HMI tags "ProLav1"
   "Lav1_Prog1_EnjIni_Cant" : Int AT 4x402562, 10 min
   "Lav1_Prog1_EnjIni_NivAg" : Int AT 4x402563, 10 min
   "Lav1_Prog1_EnjIni_Tiempo" : Int AT 4x402564, 10 min
   "Lav1_Prog1_PreLav_NivAg" : Int AT 4x402566, 10 min
   "Lav1_Prog1_PreLav_AgCaliente" : Int AT 4x402567, 10 min
   "Lav1_Prog1_Lav1_NivAg" : Int AT 4x402569, 10 min
   "Lav1_Prog1_Lav1_AgCaliente" : Int AT 4x402570, 10 min
   "Lav1_Prog1_EnjFin_Cant" : Int AT 4x402571, 10 s
   "Lav1_Prog1_Lav2_Tiempo" : Int AT 4x402617, 10 min
   "Lav1_Prog1_Lav2_NivAg" : Int AT 4x402572, 10 min
   "Lav1_Prog1_EnjFin_Tiempo" : Int AT 4x402573, 10 min
   "Lav1_Prog1_Lav2_AgCaliente" : Int AT 4x402574, 10 min
   "Lav1_Prog1_Centr_Tiempo" : Int AT 4x402575, 10 min
   "Lav1_Prog1_PreLav_Vapor" : Int AT 4x402576, 10 min
   "Lav1_Prog1_PreLav_Temperatura" : Int AT 4x402589, 10 min
   "Lav1_Prog1_Lav1_Temperatura" : Int AT 4x402591, 10 min
   "Lav1_Prog1_Lav2_Temperatura" : Int AT 4x401057, 10 min
   "Lav1_Prog1_PreLav_Tiempo" : Int AT 4x402565, 10 min
   "Lav1_Prog1_Lav1_Tiempo" : Int AT 4x402568, 10 min
   "Lav1_Prog2_EnjIni_Cant" : Int AT 4x402626, 10 min
   "Lav1_Prog2_EnjIni_NivAg" : Int AT 4x402627, 10 min
   "Lav1_Prog2_EnjIni_Tiempo" : Int AT 4x402628, 10 min
   "Lav1_Prog2_PreLav_NivAg" : Int AT 4x402630, 10 min
   "Lav1_Prog2_PreLav_AgCaliente" : Int AT 4x402631, 10 min
   "Lav1_Prog2_Lav1_NivAg" : Int AT 4x402633, 10 min
   "Lav1_Prog2_Lav1_AgCaliente" : Int AT 4x402634, 10 min
   "Lav1_Prog2_EnjFin_Cant" : Int AT 4x402635, 10 s
   "Lav1_Prog2_Lav2_Tiempo" : Int AT 4x402618, 10 min
   "Lav1_Prog2_Lav2_NivAg" : Int AT 4x402636, 10 min
   "Lav1_Prog2_EnjFin_Tiempo" : Int AT 4x402637, 10 min
   "Lav1_Prog2_Lav2_AgCaliente" : Int AT 4x402638, 10 min
   "Lav1_Prog2_Centr_Tiempo" : Int AT 4x402639, 10 min
   "Lav1_Prog2_PreLav_Vapor" : Int AT 4x402577, 10 min
   "Lav1_Prog2_PreLav_Temperatura" : Int AT 4x402592, 10 min
   "Lav1_Prog2_Lav1_Temperatura" : Int AT 4x402593, 10 min
   "Lav1_Prog2_Lav2_Temperatura" : Int AT 4x401058, 10 min
   "Lav1_Prog2_PreLav_Tiempo" : Int AT 4x402629, 10 min
   "Lav1_Prog2_Lav1_Tiempo" : Int AT 4x402632, 10 min
   "Lav1_Prog3_EnjIni_Cant" : Int AT 4x402690, 10 s
   "Lav1_Prog3_EnjIni_NivAg" : Int AT 4x402691, 10 min
   "Lav1_Prog3_EnjIni_Tiempo" : Int AT 4x402692, 10 min
   "Lav1_Prog3_PreLav_NivAg" : Int AT 4x402694, 10 min
   "Lav1_Prog3_PreLav_AgCaliente" : Int AT 4x402695, 10 min
   "Lav1_Prog3_Lav1_NivAg" : Int AT 4x402697, 10 min
   "Lav1_Prog3_Lav1_AgCaliente" : Int AT 4x402698, 10 min
   "Lav1_Prog3_EnjFin_Cant" : Int AT 4x402699, 10 min
   "Lav1_Prog3_Lav2_Tiempo" : Int AT 4x402619, 10 min
   "Lav1_Prog3_Lav2_NivAg" : Int AT 4x402700, 10 min
   "Lav1_Prog3_EnjFin_Tiempo" : Int AT 4x402701, 10 min
   "Lav1_Prog3_Lav2_AgCaliente" : Int AT 4x402702, 10 min
   "Lav1_Prog3_Centr_Tiempo" : Int AT 4x402703, 10 min
   "Lav1_Prog3_PreLav_Vapor" : Int AT 4x402579, 10 min
   "Lav1_Prog3_PreLav_Temperatura" : Int AT 4x402595, 10 min
   "Lav1_Prog3_Lav1_Temperatura" : Int AT 4x402597, 10 min
   "Lav1_Prog3_Lav2_Temperatura" : Int AT 4x401059, 10 min
   "Lav1_Prog3_PreLav_Tiempo" : Int AT 4x402693, 10 min
   "Lav1_Prog3_Lav1_Tiempo" : Int AT 4x402696, 10 min
   "Lav1_Prog4_EnjIni_Cant" : Int AT 4x402754, 10 s
   "Lav1_Prog4_EnjIni_NivAg" : Int AT 4x402755, 10 min
   "Lav1_Prog4_EnjIni_Tiempo" : Int AT 4x402756, 10 min
   "Lav1_Prog4_PreLav_NivAg" : Int AT 4x402758, 10 min
   "Lav1_Prog4_PreLav_AgCaliente" : Int AT 4x402759, 10 min
   "Lav1_Prog4_Lav1_NivAg" : Int AT 4x402761, 10 min
   "Lav1_Prog4_Lav1_AgCaliente" : Int AT 4x402762, 10 min
   "Lav1_Prog4_EnjFin_Cant" : Int AT 4x402763, 10 min
   "Lav1_Prog4_Lav2_Tiempo" : Int AT 4x402620, 10 min
   "Lav1_Prog4_Lav2_NivAg" : Int AT 4x402764, 10 min
   "Lav1_Prog4_EnjFin_Tiempo" : Int AT 4x402765, 10 min
   "Lav1_Prog4_Lav2_AgCaliente" : Int AT 4x402766, 10 min
   "Lav1_Prog4_Centr_Tiempo" : Int AT 4x402767, 10 min
   "Lav1_Prog4_PreLav_Vapor" : Int AT 4x402581, 10 min
   "Lav1_Prog4_PreLav_Temperatura" : Int AT 4x402599, 10 min
   "Lav1_Prog4_Lav1_Temperatura" : Int AT 4x402600, 10 min
   "Lav1_Prog4_Lav2_Temperatura" : Int AT 4x401060, 10 min
   "Lav1_Prog4_PreLav_Tiempo" : Int AT 4x402757, 10 min
   "Lav1_Prog4_Lav1_Tiempo" : Int AT 4x402760, 10 min
   "Lav1_Prog5_EnjIni_Cant" : Int AT 4x402818, 10 min
   "Lav1_Prog5_EnjIni_NivAg" : Int AT 4x402819, 10 min
   "Lav1_Prog5_EnjIni_Tiempo" : Int AT 4x402820, 10 min
   "Lav1_Prog5_PreLav_NivAg" : Int AT 4x402822, 10 min
   "Lav1_Prog5_PreLav_AgCaliente" : Int AT 4x402823, 10 min
   "Lav1_Prog5_Lav1_NivAg" : Int AT 4x402825, 10 min
   "Lav1_Prog5_Lav1_AgCaliente" : Int AT 4x402826, 10 min
   "Lav1_Prog5_EnjFin_Cant" : Int AT 4x402827, 10 s
   "Lav1_Prog5_Lav2_Tiempo" : Int AT 4x402621, 10 min
   "Lav1_Prog5_Lav2_NivAg" : Int AT 4x402828, 10 min
   "Lav1_Prog5_EnjFin_Tiempo" : Int AT 4x402829, 10 min
   "Lav1_Prog5_Lav2_AgCaliente" : Int AT 4x402830, 10 min
   "Lav1_Prog5_Centr_Tiempo" : Int AT 4x402831, 10 min
   "Lav1_Prog5_PreLav_Vapor" : Int AT 4x402583, 10 min
   "Lav1_Prog5_PreLav_Temperatura" : Int AT 4x402601, 10 min
   "Lav1_Prog5_Lav1_Temperatura" : Int AT 4x402603, 10 min
   "Lav1_Prog5_Lav2_Temperatura" : Int AT 4x401061, 10 min
   "Lav1_Prog5_PreLav_Tiempo" : Int AT 4x402821, 10 min
   "Lav1_Prog5_Lav1_Tiempo" : Int AT 4x402824, 10 min
   "Lav1_Prog6_EnjIni_Cant" : Int AT 4x402882, 10 min
   "Lav1_Prog6_EnjIni_NivAg" : Int AT 4x402883, 10 min
   "Lav1_Prog6_EnjIni_Tiempo" : Int AT 4x402884, 10 min
   "Lav1_Prog6_PreLav_NivAg" : Int AT 4x402886, 10 min
   "Lav1_Prog6_PreLav_AgCaliente" : Int AT 4x402887, 10 min
   "Lav1_Prog6_Lav1_NivAg" : Int AT 4x402889, 10 min
   "Lav1_Prog6_Lav1_AgCaliente" : Int AT 4x402890, 10 min
   "Lav1_Prog6_EnjFin_Cant" : Int AT 4x402891, 10 s
   "Lav1_Prog6_Lav2_Tiempo" : Int AT 4x402622, 10 min
   "Lav1_Prog6_Lav2_NivAg" : Int AT 4x402892, 10 min
   "Lav1_Prog6_EnjFin_Tiempo" : Int AT 4x402893, 10 min
   "Lav1_Prog6_Lav2_AgCaliente" : Int AT 4x402894, 10 min
   "Lav1_Prog6_Centr_Tiempo" : Int AT 4x402895, 10 min
   "Lav1_Prog6_PreLav_Vapor" : Int AT 4x402585, 10 min
   "Lav1_Prog6_PreLav_Temperatura" : Int AT 4x402605, 10 min
   "Lav1_Prog6_Lav1_Temperatura" : Int AT 4x402607, 10 min
   "Lav1_Prog6_Lav2_Temperatura" : Int AT 4x401062, 10 min
   "Lav1_Prog6_PreLav_Tiempo" : Int AT 4x402885, 10 min
   "Lav1_Prog6_Lav1_Tiempo" : Int AT 4x402888, 10 min
   "Lav1_Prog7_EnjIni_Cant" : Int AT 4x402953, 10 s
   "Lav1_Prog7_EnjIni_NivAg" : Int AT 4x402955, 10 min
   "Lav1_Prog7_EnjIni_Tiempo" : Int AT 4x402956, 10 min
   "Lav1_Prog7_PreLav_NivAg" : Int AT 4x402958, 10 min
   "Lav1_Prog7_PreLav_AgCaliente" : Int AT 4x402959, 10 min
   "Lav1_Prog7_Lav1_NivAg" : Int AT 4x402961, 10 min
   "Lav1_Prog7_Lav1_AgCaliente" : Int AT 4x402962, 10 min
   "Lav1_Prog7_EnjFin_Cant" : Int AT 4x402964, 10 min
   "Lav1_Prog7_Lav2_Tiempo" : Int AT 4x402963, 10 min
   "Lav1_Prog7_Lav2_NivAg" : Int AT 4x402965, 10 min
   "Lav1_Prog7_EnjFin_Tiempo" : Int AT 4x402966, 10 min
   "Lav1_Prog7_Lav2_AgCaliente" : Int AT 4x402967, 10 min
   "Lav1_Prog7_Centr_Tiempo" : Int AT 4x402968, 10 min
   "Lav1_Prog7_PreLav_Vapor" : Int AT 4x402969, 10 min
   "Lav1_Prog7_PreLav_Temperatura" : Int AT 4x402970, 10 min
   "Lav1_Prog7_Lav1_Temperatura" : Int AT 4x402971, 10 min
   "Lav1_Prog7_Lav2_Temperatura" : Int AT 4x401121, 10 min
   "Lav1_Prog7_PreLav_Tiempo" : Int AT 4x402957, 10 min
   "Lav1_Prog7_Lav1_Tiempo" : Int AT 4x402960, 10 min
   "Lav1_Prog8_EnjIni_Cant" : Int AT 4x402978, 10 min
   "Lav1_Prog8_EnjIni_NivAg" : Int AT 4x402979, 10 min
   "Lav1_Prog8_EnjIni_Tiempo" : Int AT 4x402980, 10 min
   "Lav1_Prog8_PreLav_NivAg" : Int AT 4x402982, 10 min
   "Lav1_Prog8_PreLav_AgCaliente" : Int AT 4x402983, 10 min
   "Lav1_Prog8_Lav1_NivAg" : Int AT 4x402985, 10 min
   "Lav1_Prog8_Lav1_AgCaliente" : Int AT 4x402986, 10 min
   "Lav1_Prog8_EnjFin_Cant" : Int AT 4x402988, 10 s
   "Lav1_Prog8_Lav2_Tiempo" : Int AT 4x402987, 10 min
   "Lav1_Prog8_Lav2_NivAg" : Int AT 4x402989, 10 min
   "Lav1_Prog8_EnjFin_Tiempo" : Int AT 4x402990, 10 min
   "Lav1_Prog8_Lav2_AgCaliente" : Int AT 4x402991, 10 min
   "Lav1_Prog8_Centr_Tiempo" : Int AT 4x402992, 10 min
   "Lav1_Prog8_PreLav_Vapor" : Int AT 4x402993, 10 min
   "Lav1_Prog8_PreLav_Temperatura" : Int AT 4x402994, 10 min
   "Lav1_Prog8_Lav1_Temperatura" : Int AT 4x402995, 10 min
   "Lav1_Prog8_Lav2_Temperatura" : Int AT 4x401186, 10 min
   "Lav1_Prog8_PreLav_Tiempo" : Int AT 4x402981, 10 min
   "Lav1_Prog8_Lav1_Tiempo" : Int AT 4x402984, 10 min
   "Lav1_Prog9_EnjIni_Cant" : Int AT 4x402996, 10 min
   "Lav1_Prog9_EnjIni_NivAg" : Int AT 4x402997, 10 min
   "Lav1_Prog9_EnjIni_Tiempo" : Int AT 4x402998, 10 min
   "Lav1_Prog9_PreLav_NivAg" : Int AT 4x403000, 10 min
   "Lav1_Prog9_PreLav_AgCaliente" : Int AT 4x403001, 10 min
   "Lav1_Prog9_Lav1_NivAg" : Int AT 4x403003, 10 min
   "Lav1_Prog9_Lav1_AgCaliente" : Int AT 4x403004, 10 min
   "Lav1_Prog9_EnjFin_Cant" : Int AT 4x403006, 10 s
   "Lav1_Prog9_Lav2_Tiempo" : Int AT 4x403005, 10 min
   "Lav1_Prog9_Lav2_NivAg" : Int AT 4x403007, 10 min
   "Lav1_Prog9_EnjFin_Tiempo" : Int AT 4x403008, 10 min
   "Lav1_Prog9_Lav2_AgCaliente" : Int AT 4x403009, 10 min
   "Lav1_Prog9_Centr_Tiempo" : Int AT 4x403010, 10 min
   "Lav1_Prog9_PreLav_Vapor" : Int AT 4x403011, 10 min
   "Lav1_Prog9_PreLav_Temperatura" : Int AT 4x403012, 10 min
   "Lav1_Prog9_Lav1_Temperatura" : Int AT 4x403013, 10 min
   "Lav1_Prog9_Lav2_Temperatura" : Int AT 4x401251, 10 min
   "Lav1_Prog9_PreLav_Tiempo" : Int AT 4x402999, 10 min
   "Lav1_Prog9_Lav1_Tiempo" : Int AT 4x403002, 10 min
   "Lav1_Prog10_EnjIni_Cant" : Int AT 4x403014, 10 min
   "Lav1_Prog10_EnjIni_NivAg" : Int AT 4x403015, 10 min
   "Lav1_Prog10_EnjIni_Tiempo" : Int AT 4x403016, 10 min
   "Lav1_Prog10_PreLav_NivAg" : Int AT 4x403018, 10 min
   "Lav1_Prog10_PreLav_AgCaliente" : Int AT 4x403019, 10 min
   "Lav1_Prog10_Lav1_NivAg" : Int AT 4x403021, 10 min
   "Lav1_Prog10_Lav1_AgCaliente" : Int AT 4x403022, 10 min
   "Lav1_Prog10_EnjFin_Cant" : Int AT 4x403024, 10 s
   "Lav1_Prog10_Lav2_Tiempo" : Int AT 4x403023, 10 min
   "Lav1_Prog10_Lav2_NivAg" : Int AT 4x403025, 10 min
   "Lav1_Prog10_EnjFin_Tiempo" : Int AT 4x403026, 10 min
   "Lav1_Prog10_Lav2_AgCaliente" : Int AT 4x403027, 10 min
   "Lav1_Prog10_Centr_Tiempo" : Int AT 4x403028, 10 min
   "Lav1_Prog10_PreLav_Vapor" : Int AT 4x403029, 10 min
   "Lav1_Prog10_PreLav_Temperatura" : Int AT 4x403030, 10 min
   "Lav1_Prog10_Lav1_Temperatura" : Int AT 4x403031, 10 min
   "Lav1_Prog10_Lav2_Temperatura" : Int AT 4x401316, 10 min
   "Lav1_Prog10_PreLav_Tiempo" : Int AT 4x403017, 10 min
   "Lav1_Prog10_Lav1_Tiempo" : Int AT 4x403020, 10 min
   "Lav1_Prog11_EnjIni_Cant" : Int AT 4x403033, 10 min
   "Lav1_Prog11_EnjIni_NivAg" : Int AT 4x403034, 10 min
   "Lav1_Prog11_EnjIni_Tiempo" : Int AT 4x403035, 10 min
   "Lav1_Prog11_PreLav_NivAg" : Int AT 4x403037, 10 min
   "Lav1_Prog11_PreLav_AgCaliente" : Int AT 4x403038, 10 min
   "Lav1_Prog11_Lav1_NivAg" : Int AT 4x403040, 10 min
   "Lav1_Prog11_Lav1_AgCaliente" : Int AT 4x403041, 10 min
   "Lav1_Prog11_EnjFin_Cant" : Int AT 4x403043, 10 s
   "Lav1_Prog11_Lav2_Tiempo" : Int AT 4x403042, 10 min
   "Lav1_Prog11_Lav2_NivAg" : Int AT 4x403044, 10 min
   "Lav1_Prog11_EnjFin_Tiempo" : Int AT 4x403045, 10 min
   "Lav1_Prog11_Lav2_AgCaliente" : Int AT 4x403046, 10 min
   "Lav1_Prog11_Centr_Tiempo" : Int AT 4x403047, 10 min
   "Lav1_Prog11_PreLav_Vapor" : Int AT 4x403048, 10 min
   "Lav1_Prog11_PreLav_Temperatura" : Int AT 4x403049, 10 min
   "Lav1_Prog11_Lav1_Temperatura" : Int AT 4x403050, 10 min
   "Lav1_Prog11_Lav2_Temperatura" : Int AT 4x401381, 10 min
   "Lav1_Prog11_PreLav_Tiempo" : Int AT 4x403036, 10 min
   "Lav1_Prog11_Lav1_Tiempo" : Int AT 4x403039, 10 min
   "Lav1_Prog12_EnjIni_Cant" : Int AT 4x403051, 10 min
   "Lav1_Prog12_EnjIni_NivAg" : Int AT 4x403052, 10 min
   "Lav1_Prog12_EnjIni_Tiempo" : Int AT 4x403053, 10 min
   "Lav1_Prog12_PreLav_NivAg" : Int AT 4x403055, 10 min
   "Lav1_Prog12_PreLav_AgCaliente" : Int AT 4x403056, 10 min
   "Lav1_Prog12_Lav1_NivAg" : Int AT 4x403058, 10 min
   "Lav1_Prog12_Lav1_AgCaliente" : Int AT 4x403059, 10 min
   "Lav1_Prog12_EnjFin_Cant" : Int AT 4x403061, 10 s
   "Lav1_Prog12_Lav2_Tiempo" : Int AT 4x403060, 10 min
   "Lav1_Prog12_Lav2_NivAg" : Int AT 4x403062, 10 min
   "Lav1_Prog12_EnjFin_Tiempo" : Int AT 4x403063, 10 min
   "Lav1_Prog12_Lav2_AgCaliente" : Int AT 4x403064, 10 min
   "Lav1_Prog12_Centr_Tiempo" : Int AT 4x403065, 10 min
   "Lav1_Prog12_PreLav_Vapor" : Int AT 4x403066, 10 min
   "Lav1_Prog12_PreLav_Temperatura" : Int AT 4x403067, 10 min
   "Lav1_Prog12_Lav1_Temperatura" : Int AT 4x403068, 10 min
   "Lav1_Prog12_Lav2_Temperatura" : Int AT 4x401382, 10 min
   "Lav1_Prog12_PreLav_Tiempo" : Int AT 4x403054, 10 min
   "Lav1_Prog12_Lav1_Tiempo" : Int AT 4x403057, 10 min
   "Lav1_Prog13_EnjIni_Cant" : Int AT 4x402091, 10 min
   "Lav1_Prog13_EnjIni_NivAg" : Int AT 4x402092, 10 min
   "Lav1_Prog13_EnjIni_Tiempo" : Int AT 4x402093, 10 min
   "Lav1_Prog13_PreLav_NivAg" : Int AT 4x402095, 10 min
   "Lav1_Prog13_PreLav_AgCaliente" : Int AT 4x402096, 10 min
   "Lav1_Prog13_Lav1_NivAg" : Int AT 4x402098, 10 min
   "Lav1_Prog13_Lav1_AgCaliente" : Int AT 4x402099, 10 min
   "Lav1_Prog13_EnjFin_Cant" : Int AT 4x402101, 10 s
   "Lav1_Prog13_Lav2_Tiempo" : Int AT 4x402100, 10 min
   "Lav1_Prog13_Lav2_NivAg" : Int AT 4x402102, 10 min
   "Lav1_Prog13_EnjFin_Tiempo" : Int AT 4x402103, 10 min
   "Lav1_Prog13_Lav2_AgCaliente" : Int AT 4x402104, 10 min
   "Lav1_Prog13_Centr_Tiempo" : Int AT 4x402105, 10 min
   "Lav1_Prog13_PreLav_Vapor" : Int AT 4x402106, 10 min
   "Lav1_Prog13_PreLav_Temperatura" : Int AT 4x402107, 10 min
   "Lav1_Prog13_Lav1_Temperatura" : Int AT 4x402108, 10 min
   "Lav1_Prog13_Lav2_Temperatura" : Int AT 4x401383, 10 min
   "Lav1_Prog13_PreLav_Tiempo" : Int AT 4x402094, 10 min
   "Lav1_Prog13_Lav1_Tiempo" : Int AT 4x402097, 10 min
   "Lav1_Prog14_EnjIni_Cant" : Int AT 4x402155, 10 min
   "Lav1_Prog14_EnjIni_NivAg" : Int AT 4x402156, 10 min
   "Lav1_Prog14_EnjIni_Tiempo" : Int AT 4x402157, 10 min
   "Lav1_Prog14_PreLav_NivAg" : Int AT 4x402159, 10 min
   "Lav1_Prog14_PreLav_AgCaliente" : Int AT 4x402160, 10 min
   "Lav1_Prog14_Lav1_NivAg" : Int AT 4x402162, 10 min
   "Lav1_Prog14_Lav1_AgCaliente" : Int AT 4x402163, 10 min
   "Lav1_Prog14_EnjFin_Cant" : Int AT 4x402165, 10 s
   "Lav1_Prog14_Lav2_Tiempo" : Int AT 4x402164, 10 min
   "Lav1_Prog14_Lav2_NivAg" : Int AT 4x402166, 10 min
   "Lav1_Prog14_EnjFin_Tiempo" : Int AT 4x402167, 10 min
   "Lav1_Prog14_Lav2_AgCaliente" : Int AT 4x402168, 10 min
   "Lav1_Prog14_Centr_Tiempo" : Int AT 4x402169, 10 min
   "Lav1_Prog14_PreLav_Vapor" : Int AT 4x402170, 10 min
   "Lav1_Prog14_PreLav_Temperatura" : Int AT 4x402171, 10 min
   "Lav1_Prog14_Lav1_Temperatura" : Int AT 4x402172, 10 min
   "Lav1_Prog14_Lav2_Temperatura" : Int AT 4x401384, 10 min
   "Lav1_Prog14_PreLav_Tiempo" : Int AT 4x402158, 10 min
   "Lav1_Prog14_Lav1_Tiempo" : Int AT 4x402161, 10 min
   "Lav1_Prog15_EnjIni_Cant" : Int AT 4x402219, 10 min
   "Lav1_Prog15_EnjIni_NivAg" : Int AT 4x402220, 10 min
   "Lav1_Prog15_EnjIni_Tiempo" : Int AT 4x402221, 10 min
   "Lav1_Prog15_PreLav_NivAg" : Int AT 4x402223, 10 min
   "Lav1_Prog15_PreLav_AgCaliente" : Int AT 4x402224, 10 min
   "Lav1_Prog15_Lav1_NivAg" : Int AT 4x402226, 10 min
   "Lav1_Prog15_Lav1_AgCaliente" : Int AT 4x402227, 10 min
   "Lav1_Prog15_EnjFin_Cant" : Int AT 4x402229, 10 s
   "Lav1_Prog15_Lav2_Tiempo" : Int AT 4x402228, 10 min
   "Lav1_Prog15_Lav2_NivAg" : Int AT 4x402230, 10 min
   "Lav1_Prog15_EnjFin_Tiempo" : Int AT 4x402231, 10 min
   "Lav1_Prog15_Lav2_AgCaliente" : Int AT 4x402232, 10 min
   "Lav1_Prog15_Centr_Tiempo" : Int AT 4x402233, 10 min
   "Lav1_Prog15_PreLav_Vapor" : Int AT 4x402234, 10 min
   "Lav1_Prog15_PreLav_Temperatura" : Int AT 4x402235, 10 min
   "Lav1_Prog15_Lav1_Temperatura" : Int AT 4x402236, 10 min
   "Lav1_Prog15_Lav2_Temperatura" : Int AT 4x401385, 10 min
   "Lav1_Prog15_PreLav_Tiempo" : Int AT 4x402222, 10 min
   "Lav1_Prog15_Lav1_Tiempo" : Int AT 4x402225, 10 min

HMI tags "Vars_Lavs_Actuales"
   "Ver_HoraFin_0" : DateTime, internal
   "Ver_HoraFin_1" : DateTime, internal
   "Ver_HoraFin_2" : DateTime, internal
   "Ver_HoraFin_3" : DateTime, internal
   "Ver_HoraFin_4" : DateTime, internal
   "Ver_HoraFin_5" : DateTime, internal
   "Ver_HoraFin_6" : DateTime, internal
   "Ver_HoraFin_7" : DateTime, internal
   "Ver_HoraFin_8" : DateTime, internal
   "Ver_HoraFin_9" : DateTime, internal
   "Ver_HoraFin_10" : DateTime, internal
   "Ver_HoraFin_11" : DateTime, internal
   "Ver_HoraFin_12" : DateTime, internal
   "Ver_HoraFin_13" : DateTime, internal
   "Ver_HoraFin_14" : DateTime, internal
   "Ver_HoraInicio_0" : DateTime, internal
   "Ver_HoraInicio_1" : DateTime, internal
   "Ver_HoraInicio_2" : DateTime, internal
   "Ver_HoraInicio_3" : DateTime, internal
   "Ver_HoraInicio_4" : DateTime, internal
   "Ver_HoraInicio_5" : DateTime, internal
   "Ver_HoraInicio_6" : DateTime, internal
   "Ver_HoraInicio_7" : DateTime, internal
   "Ver_HoraInicio_8" : DateTime, internal
   "Ver_HoraInicio_9" : DateTime, internal
   "Ver_HoraInicio_10" : DateTime, internal
   "Ver_HoraInicio_11" : DateTime, internal
   "Ver_HoraInicio_12" : DateTime, internal
   "Ver_HoraInicio_13" : DateTime, internal
   "Ver_HoraInicio_14" : DateTime, internal
   "Ver_Carga_0" : Int, internal
   "Ver_Carga_1" : Int, internal
   "Ver_Carga_2" : Int, internal
   "Ver_Carga_3" : Int, internal
   "Ver_Carga_4" : Int, internal
   "Ver_Carga_5" : Int, internal
   "Ver_Carga_6" : Int, internal
   "Ver_Carga_7" : Int, internal
   "Ver_Carga_8" : Int, internal
   "Ver_Carga_9" : Int, internal
   "Ver_Carga_10" : Int, internal
   "Ver_Carga_11" : Int, internal
   "Ver_Carga_12" : Int, internal
   "Ver_Carga_13" : Int, internal
   "Ver_Carga_14" : Int, internal
   "Ver_Programa_0" : Int, internal
   "Ver_Programa_1" : Int, internal
   "Ver_Programa_2" : Int, internal
   "Ver_Programa_3" : Int, internal
   "Ver_Programa_4" : Int, internal
   "Ver_Programa_5" : Int, internal
   "Ver_Programa_6" : Int, internal
   "Ver_Programa_7" : Int, internal
   "Ver_Programa_8" : Int, internal
   "Ver_Programa_9" : Int, internal
   "Ver_Programa_10" : Int, internal
   "Ver_Programa_11" : Int, internal
   "Ver_Programa_12" : Int, internal
   "Ver_Programa_13" : Int, internal
   "Ver_Programa_14" : Int, internal
   "Ver_HoraFin_15" : DateTime, internal
   "Ver_HoraFin_16" : DateTime, internal
   "Ver_HoraFin_17" : DateTime, internal
   "Ver_HoraFin_18" : DateTime, internal
   "Ver_HoraFin_19" : DateTime, internal
   "Ver_Programa_15" : Int, internal
   "Ver_Programa_16" : Int, internal
   "Ver_Programa_17" : Int, internal
   "Ver_Programa_18" : Int, internal
   "Ver_Programa_19" : Int, internal
   "Ver_Carga_15" : Int, internal
   "Ver_Carga_16" : Int, internal
   "Ver_Carga_17" : Int, internal
   "Ver_Carga_18" : Int, internal
   "Ver_Carga_19" : Int, internal
   "Ver_HoraInicio_15" : DateTime, internal
   "Ver_HoraInicio_16" : DateTime, internal
   "Ver_HoraInicio_17" : DateTime, internal
   "Ver_HoraInicio_18" : DateTime, internal
   "Ver_HoraInicio_19" : DateTime, internal
   "Ver_Cli_Str_0" : WString[64], internal
   "Ver_Cli_Str_1" : WString[64], internal
   "Ver_Cli_Str_2" : WString[64], internal
   "Ver_Cli_Str_3" : WString[64], internal
   "Ver_Cli_Str_4" : WString[64], internal
   "Ver_Cli_Str_5" : WString[64], internal
   "Ver_Cli_Str_6" : WString[64], internal
   "Ver_Cli_Str_7" : WString[64], internal
   "Ver_Cli_Str_8" : WString[64], internal
   "Ver_Cli_Str_9" : WString[64], internal
   "Ver_Cli_Str_10" : WString[64], internal
   "Ver_Cli_Str_11" : WString[64], internal
   "Ver_Cli_Str_12" : WString[64], internal
   "Ver_Cli_Str_13" : WString[64], internal
   "Ver_Cli_Str_14" : WString[64], internal
   "Ver_Cli_Str_15" : WString[64], internal
   "Ver_Cli_Str_16" : WString[64], internal
   "Ver_Cli_Str_17" : WString[64], internal
   "Ver_Cli_Str_18" : WString[64], internal
   "Ver_Cli_Str_19" : WString[64], internal
   "Ver_Operador_Str_0" : WString[64], internal
   "Ver_Operador_Str_1" : WString[64], internal
   "Ver_Operador_Str_2" : WString[64], internal
   "Ver_Operador_Str_3" : WString[64], internal
   "Ver_Operador_Str_4" : WString[64], internal
   "Ver_Operador_Str_5" : WString[64], internal
   "Ver_Operador_Str_6" : WString[64], internal
   "Ver_Operador_Str_7" : WString[64], internal
   "Ver_Operador_Str_8" : WString[64], internal
   "Ver_Operador_Str_9" : WString[64], internal
   "Ver_Operador_Str_10" : WString[64], internal
   "Ver_Operador_Str_11" : WString[64], internal
   "Ver_Operador_Str_12" : WString[64], internal
   "Ver_Operador_Str_13" : WString[64], internal
   "Ver_Operador_Str_14" : WString[64], internal
   "Ver_Operador_Str_15" : WString[64], internal
   "Ver_Operador_Str_16" : WString[64], internal
   "Ver_Operador_Str_17" : WString[64], internal
   "Ver_Operador_Str_18" : WString[64], internal
   "Ver_Operador_Str_19" : WString[64], internal
   "Ver_IDList" : Int, internal
   "Ver_Anim_Boton" : Int, internal
   "Ver_CicloValido_0" : Bool, internal
   "Ver_CicloValido_1" : Bool, internal
   "Ver_CicloValido_2" : Bool, internal
   "Ver_CicloValido_3" : Bool, internal
   "Ver_CicloValido_4" : Bool, internal
   "Ver_CicloValido_5" : Bool, internal
   "Ver_CicloValido_6" : Bool, internal
   "Ver_CicloValido_7" : Bool, internal
   "Ver_CicloValido_8" : Bool, internal
   "Ver_CicloValido_9" : Bool, internal
   "Ver_CicloValido_10" : Bool, internal
   "Ver_CicloValido_11" : Bool, internal
   "Ver_CicloValido_12" : Bool, internal
   "Ver_CicloValido_13" : Bool, internal
   "Ver_CicloValido_14" : Bool, internal
   "Ver_CicloValido_15" : Bool, internal
   "Ver_CicloValido_16" : Bool, internal
   "Ver_CicloValido_17" : Bool, internal
   "Ver_CicloValido_18" : Bool, internal
   "Ver_CicloValido_19" : Bool, internal
   "Ver_Programa_X" : Int, internal
   "Ver_Operador_Int_X" : Int, internal
   "Ver_HoraInicio_X" : DateTime, internal
   "Ver_HoraFin_X" : DateTime, internal
   "Ver_Cli1_Str_X" : Int, internal
   "Ver_CicloValido_X" : Int, internal
   "Ver_Carga_X" : Int, internal
   "Ver_Editor_X" : Bool, internal
   "Ver_DIA_X" : DateTime, internal
   "Ver_Cli2_Str_X" : Int, internal
   "Ver_Cli3_Str_X" : Int, internal
   "Ver_Cli_Str_X" : WString[64], internal
   "Ver_Operador_WStr_X" : WString[64], internal
   "Ver_Programa_X_ans" : Int, internal
   "Ver_Operador_Int_X_ans" : Int, internal
   "Ver_HoraFin_X_ans" : DateTime, internal
   "Ver_Cli1_Str_X_ans" : Int, internal
   "Ver_Cli2_Str_X_ans" : Int, internal
   "Ver_Cli3_Str_X_ans" : Int, internal
   "Ver_DIA_X_ans" : DateTime, internal
   "Ver_CicloValido_X_ans" : Int, internal
   "Ver_Carga_X_ans" : Int, internal
   "Ver_HoraInicio_X_ans" : DateTime, internal
   "Ver_DIA_XP" : DateTime, internal
   "Ver_DIA_X_ansP" : DateTime, internal

HMI tags "Informes"
   "Inf_Mes" : Int, internal
   "Inf_Desde" : DateTime, internal
   "Inf_Hasta" : DateTime, internal
   "Inf_Ano" : Int, internal
   "InfP_Ano" : Int, internal
   "InfP_Desde" : DateTime, internal
   "InfP_Hasta" : DateTime, internal
   "InfP_Mes" : Int, internal

HMI tags "Lista Indices"
   "Idx_ID" : Int AT %DB1.DBW0
   "Idx_Name" : Int AT %DB1.DBX0.0
   "Idx_ID_1" : Int, internal
   "Idx_ID_Cambiar" : Int, internal
   "Idx_ID_Nuevo" : Int, internal
   "Idx_Name_1" : Int, internal
   "Idx_Name_2" : Int, internal
   "Idx_Name_3" : Int, internal
   "Idx_Name_4" : Int, internal
   "Idx_Name_5" : Int, internal
   "Idx_Name_Cambiar" : Int, internal
   "Idx_Name_Nuevo" : Int, internal
   "Idx_ID_2" : Int, internal
   "Idx_ID_3" : Int, internal
   "Idx_ID_4" : Int, internal
   "Idx_ID_5" : Int, internal

HMI tags "Generales"
   "_Prog_Centr_Tiempo" : UInt, internal
   "_Prog_EnjFin_Cant" : UInt, internal
   "_Prog_EnjFin_Tiempo" : UInt, internal
   "_Prog_EnjIni_Cant" : UInt, internal
   "_Prog_EnjIni_NivAg" : UInt, internal
   "_Prog_EnjIni_Tiempo" : UInt, internal
   "_Prog_Lav1_AgCaliente" : UInt, internal
   "_Prog_Lav1_NivAg" : UInt, internal
   "_Prog_Lav1_Temperatura" : UInt, internal
   "_Prog_Lav1_Tiempo" : UInt, internal
   "_Prog_Lav2_AgCaliente" : UInt, internal
   "_Prog_Lav2_NivAg" : UInt, internal
   "_Prog_Lav2_Temperatura" : UInt, internal
   "_Prog_Lav2_Tiempo" : UInt, internal
   "_Prog_PreLav_AgCaliente" : UInt, internal
   "_Prog_PreLav_NivAg" : UInt, internal
   "_Prog_PreLav_Temperatura" : UInt, internal
   "_Prog_PreLav_Tiempo" : UInt, internal
   "_Prog_PreLav_Vapor" : UInt, internal
   "_Prog_aModifBraun" : UInt, internal
   "_Prog_aModifGirbau" : UInt, internal
   "_Prog_Prueba" : Int AT 4x403187, 1 s
   "_errorNum1" : UInt, internal
   "_errorNum2" : UInt, internal
   "_errorNum3" : UInt, internal
   "_errorNum4" : UInt, internal

discrete alarms
   1: 'Planch1: Falla de sensor Izquierdo', class Errors, trigger "Ala-Disp-W0" bit 8
   2: 'Planch1: Falla de sensor Central', class Errors, trigger "Ala-Disp-W0" bit 9
   3: 'Planch1: Falla de sensor Derecho', class Errors, trigger "Ala-Disp-W0" bit 10
   4: 'Planch2: Falla de sensor Izquierdo', class Errors, trigger "Ala-Disp-W0" bit 11
   5: 'Planch2: Falla de sensor Central', class Errors, trigger "Ala-Disp-W0" bit 12
   6: 'Planch2: Falla de sensor Derecho', class Errors, trigger "Ala-Disp-W0" bit 13
   7: 'Res-6', class Errors, trigger "Ala-Disp-W0" bit 14
   8: 'Res-7', class Errors, trigger "Ala-Disp-W0" bit 15
   9: 'Res-8', class Errors, trigger "Ala-Disp-W0" bit 0
   10: 'Res-9', class Errors, trigger "Ala-Disp-W0" bit 1
   11: 'Res-10', class Errors, trigger "Ala-Disp-W0" bit 2
   12: 'Res-11', class Errors, trigger "Ala-Disp-W0" bit 3
   13: 'Res-12', class Errors, trigger "Ala-Disp-W0" bit 4
   14: 'Res-13', class Errors, trigger "Ala-Disp-W0" bit 5
   15: 'Res-14', class Errors, trigger "Ala-Disp-W0" bit 6
   16: 'Res-15', class Errors, trigger "Ala-Disp-W0" bit 7
   17: 'Res-16', class Errors, trigger "Ala-Disp-W1" bit 8
   18: 'Res-17', class Errors, trigger "Ala-Disp-W1" bit 9
   19: 'Res-18', class Errors, trigger "Ala-Disp-W1" bit 10
   20: 'Res-19', class Errors, trigger "Ala-Disp-W1" bit 11
   21: 'Res-20', class Errors, trigger "Ala-Disp-W1" bit 12
   22: 'Res-21', class Errors, trigger "Ala-Disp-W1" bit 13
   23: 'Res-22', class Errors, trigger "Ala-Disp-W1" bit 14
   24: 'Res-23', class Errors, trigger "Ala-Disp-W1" bit 15
   25: 'Res-24', class Errors, trigger "Ala-Disp-W1" bit 0
   26: 'Res-25', class Errors, trigger "Ala-Disp-W1" bit 1
   27: 'Res-26', class Errors, trigger "Ala-Disp-W1" bit 2
   28: 'Res-27', class Errors, trigger "Ala-Disp-W1" bit 3
   29: 'Res-28', class Errors, trigger "Ala-Disp-W1" bit 4
   30: 'Res-29', class Errors, trigger "Ala-Disp-W1" bit 5
   31: 'Res-30', class Errors, trigger "Ala-Disp-W1" bit 6
   32: 'Res-31', class Errors, trigger "Ala-Disp-W1" bit 7

text list "Lista de textos_1": 1 'Domingo'; 2 'Lunes'; 3 'Martes'; 4 'Miercoles'; 5 'Jueves'; 6 'Viernes'; 7 'Sabado'

text list "Operadores_Lavadora": 0 ''; 1 'BENITEZ M'; 2 'MARTINEZ C'; 3 'SALINAS C'; 4 'BOGARIN M'; 5 'MARTINEZ A'; 6 'RODAS A'; 7 'TELLO C'; 8 'MARCATO S'

text list "Clientes": 1 'S CENTRO-BLANCO'; 2 'BASF'; 3 'S IPAM-BLANCO'; 4 'S IPAM-VERDE'; 5 'CTC-BLANCO'; 6 'CTC-GUARDAPOLVOS'; 7 'CDI DEL NORTE'; 8 'ELAS-BLANCO'; 9 'ELAS-GUARDAPOLVOS'; 10 'CATAMARCA APART'; 11 '1495 APART'; 12 'GAUROS'; 13 'GO ALTO-BLANCO'; 14 'GO ALTO-GUARDAPOLVOS'; 15 'GAMMA'; 16 'H MAYORAL'; 17 'HECA'; 18 'SANTA ROSA HOGAR'; 19 'HPR-BLANCO'; 20 'HPR-VERDE'; 21 'HPR-GUARDAPOLVO'; 22 'REAL ROSARIO HOSTEL'; 23 'INECO-BLANCO'; 24 'INECO-GUARDAPOLVOS'; 25 'ICR-BLANCO'; 26 'ICR-VERDE'; 27 'ICR-GUARDAPOLVOS'; 28 'VAPOX LAB'; 29 'LIMPAR'; 30 'MANTELERIA BLANCA ALQ'; 31 'MANTELERIA NEGRA ALQ'; 32 'MARTIN CIRIBENI'; 33 'ROSTOWER'; 34 'UOM-BLANCO'; 35 'UOM-VERDE'; 36 'RGOLF TOALLONES'; 37 'HOWARD J HOTEL'; 38 'S BRITANICO'; 39 'S NIÑOS'; 40 'S MAPACI'; 41 'S PARQUE'; 42 'S PLAZA'; 43 'SWIFT-BLANCO'; 44 'SWIFT-VERDE'; 45 'SWIFT-GRASA'; 46 'UMMA'; 47 'ZONA NORTE H'; 48 'TOALLAS'; 49 'FRAZADAS'; 50 'RELAVADOS-BLANCO'; 51 'RELAVADO-VERDE'; 52 'S CENTRO-V'; 53 'S NIÑOS-V'; 54 'MAPACI-V'; 55 'PLAZA-V'; 56 'PARQUE GUARD'; 57 'SILV PARQ'; 58 'SILV ICR'; 59 'SILV NINOS'; 60 'BATA LILA ALQ'; 61 'GAMMA-V'; 62 'PALADINI'; 63 'PARQUE-V'; 64 'BRITANICO-V'; 65 'GTE BLANCO'; 66 'GTE AMARILLO'; 67 'MANGAS'; 68 'MAM TERRAG'; 69 'HPR AMBOS COLOR'; 70 'ICR AMBOS COLOR'; 71 'SILV CARRASCO'; 72 'SILV ALBERDI'; 73 'SILV SAEZ PEÑA'; 74 'SILV SIES'; 75 'SILV H NINOS'; 76 'SILV M MARTIN'; 77 'PARQUE AMBO BLANC'; 78 'LIMPAR GRASAS'; 79 'ALFOMBRAS'; 80 ''; 81 ''; 82 ''; 83 ''; 84 ''; 85 ''; 86 ''

screen "Principal" 1366x768, template "Pulsadores"
   Rectangle "Rectángulo_12" at 26,396 size 259x170
      Appearance <- "Lav3_Alarma"
   Rectangle "Rectángulo_8" at 26,217 size 259x170
      Appearance <- "Lav2_Alarma"
   Rectangle "Rectángulo_10" at 26,38 size 259x170
      Appearance <- "Lav1_Alarma"
   TrendView "Visor de curvas_1" at 305,70 size 977x527
   TextField "Campo de texto_1" at 497,667 size 107x33; Text 'Objetivo'
   TextField "Campo de texto_2" at 766,667 size 98x33; Text 'Avance'
   TextField "Campo de texto_3" at 502,16 size 164x36; Text 'PLANCHAS'
   Circle "Círculo_1" at 1307,127 size 34x34
      Appearance <- "Planchadora1_EstadoSsIzq"
   Circle "Círculo_2" at 1307,188 size 34x34
      Appearance <- "Planchadora1_EstadoSSMed"
   Circle "Círculo_3" at 1307,249 size 34x34
      Appearance <- "Planchadora1_EstadoSsDer"
   TextField "Campo de texto_10" at 1317,99 size 15x22; Text 'Text'
   TextField "Campo de texto_11" at 1302,95 size 44x27; Text 'SNS'
   TextField "Campo de texto_12" at 1310,163 size 29x22; Text 'Izq'
   TextField "Campo de texto_13" at 1306,223 size 36x22; Text 'Med'
   TextField "Campo de texto_14" at 1307,283 size 32x22; Text 'Der'
   TextField "Campo de texto_15" at 1192,279 size 15x22; Text 'Text'
   Switch "Interruptor_6" at 720,8 size 111x52; TextOn 'CHIC 1 MARCHA'; CaptionText 'OK'; TextOff 'CHIC 1 PARADA'
      ProcessValue <- "MaqEnProd"
   IOField "Campo ES_46" at 1065,1 size 300x37; FormatPattern 9999999999999999999999999999999999999999
      ProcessValue <- "Planchadora1_FechaHoraPLC"
   Button "Botón_2882" at 1205,720 size 161x48; TextOff 'ALARMAS'
      on Click: ActivateScreen("Alarmas", 0)
   TextField "Campo de texto_17" at 1186,405 size 15x22; Text 'Text'
   Switch "Interruptor_8" at 876,8 size 111x52; TextOn 'CHIC 2 MARCHA'; CaptionText 'OK'; TextOff 'CHIC 2 PARADA'
      ProcessValue <- "Plan2EnProd"
   TextField "Campo de texto_5" at 70,0 size 187x36; Text 'LAVADORAS'
   Rectangle "Rectángulo_9" at 40,295 size 88x38
      Appearance <- "Lav2_EnCiclo"
   IOField "Campo ES_9" at 70,291 size 57x41; FormatPattern FF
      ProcessValue <- "Lav2_Programa"
   TextField "Campo de texto_30" at 60,222 size 45x68; Text '2'
   Rectangle "Rectángulo_11" at 40,116 size 88x38
      Appearance <- "Lav1_EnCiclo"
   TextField "Campo de texto_31" at 138,128 size 32x20; Text 'Op:'
   TextField "Campo de texto_32" at 41,109 size 26x48; Text 'P'
   IOField "Campo ES_12" at 72,112 size 57x41; FormatPattern FF
      ProcessValue <- "Lav1_Programa"
   TextField "Campo de texto_33" at 131,108 size 62x22; Text 'Carga:'
   IOField "Campo ES_13" at 189,110 size 76x18; FormatPattern 99999; Unit  Kg
      ProcessValue <- "Lav1_CantRopa"
   TextField "Campo de texto_35" at 60,43 size 45x68; Text '1'
   Rectangle "Rectángulo_13" at 40,474 size 88x38
      Appearance <- "Lav3_EnCiclo"
   TextField "Campo de texto_37" at 41,467 size 26x48; Text 'P'
   IOField "Campo ES_15" at 71,471 size 57x41; FormatPattern FF
      ProcessValue <- "Lav3_Programa"
   TextField "Campo de texto_40" at 60,401 size 45x68; Text '3'
   TextField "Campo de texto_6" at 41,288 size 26x48; Text 'P'
   IOField "Campo ES_6" at 170,129 size 97x18; FormatPattern ????????????????????????????????????????????????????????????????
      ProcessValue <- "Lav1_Operador_Str"
   Rectangle "Rectángulo_1" at 26,572 size 259x170
      Appearance <- "Lav4_Alarma"
   Rectangle "Rectángulo_17" at 40,650 size 88x38
      Appearance <- "Lav4_EnCiclo"
   TextField "Campo de texto_8" at 41,643 size 26x48; Text 'P'
   IOField "Campo ES_11" at 71,646 size 57x41; FormatPattern FF
      ProcessValue <- "Lav4_Programa"
   TextField "Campo de texto_25" at 60,577 size 45x68; Text '4'
   TextField "Campo de texto_26" at 121,48 size 22x61; Text 'Clientes'
   IOField "Campo ES_18" at 144,47 size 129x21; FormatPattern ????????????????????????????????????????????????????????????????
      ProcessValue <- "Lav1_Cli_0_Str"
   IOField "Campo ES_19" at 144,66 size 129x21; FormatPattern ????????????????????????????????????????????????????????????????
      ProcessValue <- "Lav1_Cli_1_Str"
   IOField "Campo ES_20" at 144,85 size 129x21; FormatPattern ????????????????????????????????????????????????????????????????
      ProcessValue <- "Lav1_Cli_2_Str"
   TextField "Campo de texto_7" at 138,306 size 32x20; Text 'Op:'
   TextField "Campo de texto_24" at 131,286 size 62x22; Text 'Carga:'
   IOField "Campo ES_7" at 189,288 size 76x18; FormatPattern 99999; Unit  Kg
      ProcessValue <- "Lav2_CantRopa"
   IOField "Campo ES_8" at 170,307 size 97x18; FormatPattern ????????????????????????????????????????????????????????????????
      ProcessValue <- "Lav2_Operador_Str"
   TextField "Campo de texto_27" at 121,227 size 23x65; Text 'Clientes'
   IOField "Campo ES_10" at 144,225 size 129x21; FormatPattern ????????????????????????????????????????????????????????????????
      ProcessValue <- "Lav2_Cli_0_Str"
   IOField "Campo ES_14" at 144,244 size 129x21; FormatPattern ????????????????????????????????????????????????????????????????
      ProcessValue <- "Lav2_Cli_1_Str"
   IOField "Campo ES_16" at 144,263 size 129x21; FormatPattern ????????????????????????????????????????????????????????????????
      ProcessValue <- "Lav2_Cli_2_Str"
   TextField "Campo de texto_28" at 138,486 size 32x20; Text 'Op:'
   TextField "Campo de texto_29" at 131,466 size 62x22; Text 'Carga:'
   IOField "Campo ES_17" at 189,468 size 76x18; FormatPattern 99999; Unit  Kg
      ProcessValue <- "Lav3_CantRopa"
   IOField "Campo ES_21" at 170,487 size 97x18; FormatPattern ????????????????????????????????????????????????????????????????
      ProcessValue <- "Lav3_Operador_Str"
   IOField "Campo ES_22" at 144,405 size 129x21; FormatPattern ????????????????????????????????????????????????????????????????
      ProcessValue <- "Lav3_Cli_0_Str"
   IOField "Campo ES_23" at 144,424 size 129x21; FormatPattern ????????????????????????????????????????????????????????????????
      ProcessValue <- "Lav3_Cli_1_Str"
   IOField "Campo ES_24" at 144,443 size 129x21; FormatPattern ????????????????????????????????????????????????????????????????
      ProcessValue <- "Lav3_Cli_2_Str"
   TextField "Campo de texto_36" at 138,660 size 32x20; Text 'Op:'
   TextField "Campo de texto_38" at 131,640 size 62x22; Text 'Carga:'
   IOField "Campo ES_25" at 189,642 size 76x18; FormatPattern 99999; Unit  Kg
      ProcessValue <- "Lav4_CantRopa"
   IOField "Campo ES_26" at 170,661 size 97x18; FormatPattern ????????????????????????????????????????????????????????????????
      ProcessValue <- "Lav4_Operador_Str"
   IOField "Campo ES_27" at 144,580 size 129x21; FormatPattern ????????????????????????????????????????????????????????????????
      ProcessValue <- "Lav4_Cli_0_Str"
   IOField "Campo ES_28" at 144,599 size 129x21; FormatPattern ????????????????????????????????????????????????????????????????
      ProcessValue <- "Lav4_Cli_1_Str"
   IOField "Campo ES_29" at 144,618 size 129x21; FormatPattern ????????????????????????????????????????????????????????????????
      ProcessValue <- "Lav4_Cli_2_Str"
   Circle "Círculo_4" at 1307,415 size 34x34
      Appearance <- "Planchadora2_EstadoSsIzq"
   Circle "Círculo_5" at 1307,476 size 34x34
      Appearance <- "Planchadora2_EstadoSSMed"
   Circle "Círculo_6" at 1307,537 size 34x34
      Appearance <- "Planchadora2_EstadoSsDer"
   TextField "Campo de texto_16" at 1317,387 size 15x22; Text 'Text'
   TextField "Campo de texto_18" at 1302,383 size 44x27; Text 'SNS'
   TextField "Campo de texto_19" at 1310,451 size 29x22; Text 'Izq'
   TextField "Campo de texto_20" at 1306,511 size 36x22; Text 'Med'
   TextField "Campo de texto_21" at 1307,571 size 32x22; Text 'Der'
   TextField "Campo de texto_9" at 51,157 size 64x20; Text 'INICIO'
   TextField "Campo de texto_22" at 155,157 size 115x20; Text 'FIN ESTIMADO'
   IOField "Campo ES_3" at 58,177 size 30x16; FormatPattern FF; Unit :
      ProcessValue <- "Lav1_FchIni_Hr"
   IOField "Campo ES_30" at 88,177 size 24x16; FormatPattern FF
      ProcessValue <- "Lav1_FchIni_Min"
   IOField "Campo ES_31" at 186,177 size 75x16; FormatPattern 9999999999999999999999999999999999999999
      ProcessValue <- "Lav1_FinEstimado_Panel"
   TextField "Campo de texto_34" at 121,406 size 22x61; Text 'Clientes'
   TextField "Campo de texto_39" at 121,580 size 22x61; Text 'Clientes'
   TextField "Campo de texto_41" at 51,334 size 64x20; Text 'INICIO'
   TextField "Campo de texto_42" at 155,334 size 115x20; Text 'FIN ESTIMADO'
   IOField "Campo ES_32" at 58,354 size 30x16; FormatPattern FF; Unit :
      ProcessValue <- "Lav2_FchIni_Hr"
   IOField "Campo ES_33" at 88,354 size 24x16; FormatPattern FF
      ProcessValue <- "Lav2_FchIni_Min"
   IOField "Campo ES_34" at 186,354 size 75x16; FormatPattern 9999999999999999999999999999999999999999
      ProcessValue <- "Lav2_FinEstimado_Panel"
   TextField "Campo de texto_43" at 51,513 size 64x20; Text 'INICIO'
   TextField "Campo de texto_44" at 155,513 size 115x20; Text 'FIN ESTIMADO'
   IOField "Campo ES_35" at 58,533 size 30x16; FormatPattern FF; Unit :
      ProcessValue <- "Lav3_FchIni_Hr"
   IOField "Campo ES_36" at 88,533 size 24x16; FormatPattern FF
      ProcessValue <- "Lav3_FchIni_Min"
   IOField "Campo ES_37" at 186,533 size 75x16; FormatPattern 9999999999999999999999999999999999999999
      ProcessValue <- "Lav3_FinEstimado_Panel"
   TextField "Campo de texto_45" at 51,690 size 64x20; Text 'INICIO'
   TextField "Campo de texto_46" at 155,690 size 115x20; Text 'FIN ESTIMADO'
   IOField "Campo ES_38" at 58,710 size 30x16; FormatPattern FF; Unit :
      ProcessValue <- "Lav4_FchIni_Hr"
   IOField "Campo ES_39" at 88,710 size 24x16; FormatPattern FF
      ProcessValue <- "Lav4_FchIni_Min"
   IOField "Campo ES_40" at 186,710 size 75x16; FormatPattern 9999999999999999999999999999999999999999
      ProcessValue <- "Lav4_FinEstimado_Panel"
   Button "Botón_333" at 565,720 size 161x48; TextOff 'REGISTROS DE LAVADOS'
      on Click: ActivateScreen("Lavados_Actuales", 0); "S403_ActDia"()
   Button "Botón_14456" at 1045,720 size 161x48; TextOff 'CONFIGURACION'
      on Click: ActivateScreen("Configuracion", 0)
   Button "Botón_4" at 129,580 size 140x154; TextOff 'Text'
      on Click: ActivateScreen("Lavados_Actuales", 0); SetTag("Ver_IDList", 0); SetTag("Ver_Anim_Boton", 4); "S403_ActDia"(); "S400_ActListLav"(4)
   Button "Botón_5578" at 39,581 size 92x94; TextOff 'Text'
      on Click: ActivateScreen("Prog_Lav4_0", 0)
   Button "Botón_6" at 129,404 size 140x154; TextOff 'Text'
      on Click: ActivateScreen("Lavados_Actuales", 0); SetTag("Ver_IDList", 0); SetTag("Ver_Anim_Boton", 3); "S403_ActDia"(); "S400_ActListLav"(3)
   Button "Botón_8" at 129,225 size 140x154; TextOff 'Text'
      on Click: ActivateScreen("Lavados_Actuales", 0); SetTag("Ver_IDList", 0); SetTag("Ver_Anim_Boton", 2); "S403_ActDia"(); "S400_ActListLav"(2)
   Button "Botón_10" at 129,46 size 148x154; TextOff 'Text'
      on Click: ActivateScreen("Lavados_Actuales", 0); SetTag("Ver_IDList", 0); SetTag("Ver_Anim_Boton", 1); "S403_ActDia"(); "S400_ActListLav"(1)
   Button "Botón_7" at 39,406 size 92x94; TextOff 'Text'
      on Click: ActivateScreen("Prog_Lav3_0", 0)
   Button "Botón_9" at 38,226 size 92x94; TextOff 'Text'
      on Click: ActivateScreen("Prog_Lav2_0", 0)
   Button "Botón_11" at 38,47 size 92x94; TextOff 'Text'
      on Click: ActivateScreen("Prog_Lav1_0", 0)
   Button "Botón_13865" at 405,720 size 161x48; TextOff 'INFORMES'
      on Click: ActivateScreen("Informes", 0); "S403_ActDia"()
   Button "Botón_2574" at 725,720 size 161x48; TextOff 'INDICES Y CLIENTES'
      on Click: ActivateScreen("RegyClientes", 0); SetTag("ID_1", 1); "S103_ActualizarLista"(); "S201_ActualizarSupervisor"(); "S303_ActualizarListaOp"(); SetTag("Idx_ID_1", 1); "I103_ActualizarIndice"()
   TextField "Campo de texto_4" at 1002,667 size 153x33; Text 'Tiempo Real'
   IOField "Campo ES_1" at 436,620 size 134x47; FormatPattern 99999999999999999999
      ProcessValue <- "Indices_objetivo"
   IOField "Campo ES_2" at 700,620 size 134x47; FormatPattern 99999999999999999999
      ProcessValue <- "Indices_avance"
   IOField "Campo ES_4" at 964,620 size 134x47; FormatPattern 99999999999999999999
      ProcessValue <- "Indices_real"
   IOField "Campo ES_5" at 836,620 size 94x47; FormatPattern 99; Unit %
      ProcessValue <- "Indices_avance_100"
   IOField "Campo ES_41" at 572,620 size 94x47; FormatPattern 99; Unit %
      ProcessValue <- "Indices_objetivo_100"
   IOField "Campo ES_42" at 1100,620 size 94x47; FormatPattern 99; Unit %
      ProcessValue <- "Indices_avance_real_100"
   IOField "Campo ES_43" at 300,620 size 118x47; FormatPattern 99
      ProcessValue <- "Planchadora1_SumaOperario"
   TextField "Campo de texto_23" at 297,667 size 120x33; Text 'Operarios'
   Button "Botón_12" at 1204,611 size 161x48; TextOff 'TENDENCIA'
      on Click: ActivateScreen("Tendencias", 0)
   Button "Botón_1" at 885,720 size 161x48; TextOff 'PROCESOS'
      on Click: ActivateScreen("Procesos", 0)
   Button "Botón_2" at 293,720 size 113x48; TextOff 'ACT HORA LAVS'
      on Click: "SA3_Act_HoraFinEstPrincLav1"(); "SA3_Act_HoraFinEstPrincLav2"(); "SA3_Act_HoraFinEstPrincLav3"(); "SA3_Act_HoraFinEstPrincLav4"()

screen "Horario_Supervisor" 1366x768, template "Pulsadores"
   IOField "Campo ES_1" at 188,447 size 86x32; FormatPattern 99999999999999999999
      ProcessValue <- "Planchadora1_Supervisores{1}_Diadelasemana{1}_Entrda"
   IOField "Campo ES_2" at 294,447 size 86x32; FormatPattern 99999999999999999999
      ProcessValue <- "Planchadora1_Supervisores{1}_Diadelasemana{1}_Salida"
   IOField "Campo ES_3" at 188,173 size 86x32; FormatPattern 99999999999999999999
      ProcessValue <- "Planchadora1_Supervisores{1}_Diadelasemana{2}_Entrda"
   IOField "Campo ES_4" at 294,173 size 86x32; FormatPattern 99999999999999999999
      ProcessValue <- "Planchadora1_Supervisores{1}_Diadelasemana{2}_Salida"
   IOField "Campo ES_5" at 188,219 size 86x32; FormatPattern 99999999999999999999
      ProcessValue <- "Planchadora1_Supervisores{1}_Diadelasemana{3}_Entrda"
   IOField "Campo ES_6" at 294,219 size 86x32; FormatPattern 99999999999999999999
      ProcessValue <- "Planchadora1_Supervisores{1}_Diadelasemana{3}_Salida"
   IOField "Campo ES_7" at 188,265 size 86x32; FormatPattern 99999999999999999999
      ProcessValue <- "Planchadora1_Supervisores{1}_Diadelasemana{4}_Entrda"
   IOField "Campo ES_8" at 294,265 size 86x32; FormatPattern 99999999999999999999
      ProcessValue <- "Planchadora1_Supervisores{1}_Diadelasemana{4}_Salida"
   IOField "Campo ES_9" at 188,311 size 86x32; FormatPattern 99999999999999999999
      ProcessValue <- "Planchadora1_Supervisores{1}_Diadelasemana{5}_Entrda"
   IOField "Campo ES_10" at 294,311 size 86x32; FormatPattern 99999999999999999999
      ProcessValue <- "Planchadora1_Supervisores{1}_Diadelasemana{5}_Salida"
   IOField "Campo ES_11" at 188,357 size 86x32; FormatPattern 99999999999999999999
      ProcessValue <- "Planchadora1_Supervisores{1}_Diadelasemana{6}_Entrda"
   IOField "Campo ES_12" at 294,357 size 86x32; FormatPattern 99999999999999999999
      ProcessValue <- "Planchadora1_Supervisores{1}_Diadelasemana{6}_Salida"
   IOField "Campo ES_13" at 188,403 size 86x32; FormatPattern 99999999999999999999
      ProcessValue <- "Planchadora1_Supervisores{1}_Diadelasemana{7}_Entrda"
   IOField "Campo ES_14" at 294,403 size 86x32; FormatPattern 99999999999999999999
      ProcessValue <- "Planchadora1_Supervisores{1}_Diadelasemana{7}_Salida"
   IOField "Campo ES_15" at 479,447 size 86x32; FormatPattern 99999999999999999999
      ProcessValue <- "Planchadora1_Supervisores{2}_Diadelasemana{1}_Entrda"
   IOField "Campo ES_16" at 589,447 size 86x32; FormatPattern 99999999999999999999
      ProcessValue <- "Planchadora1_Supervisores{2}_Diadelasemana{1}_Salida"
   IOField "Campo ES_17" at 479,173 size 86x32; FormatPattern 99999999999999999999
      ProcessValue <- "Planchadora1_Supervisores{2}_Diadelasemana{2}_Entrda"
   IOField "Campo ES_18" at 589,173 size 86x32; FormatPattern 99999999999999999999
      ProcessValue <- "Planchadora1_Supervisores{2}_Diadelasemana{2}_Salida"
   IOField "Campo ES_19" at 479,219 size 86x32; FormatPattern 99999999999999999999
      ProcessValue <- "Planchadora1_Supervisores{2}_Diadelasemana{3}_Entrda"
   IOField "Campo ES_20" at 589,219 size 86x32; FormatPattern 99999999999999999999
      ProcessValue <- "Planchadora1_Supervisores{2}_Diadelasemana{3}_Salida"
   IOField "Campo ES_21" at 479,265 size 86x32; FormatPattern 99999999999999999999
      ProcessValue <- "Planchadora1_Supervisores{2}_Diadelasemana{4}_Entrda"
   IOField "Campo ES_22" at 589,265 size 86x32; FormatPattern 99999999999999999999
      ProcessValue <- "Planchadora1_Supervisores{2}_Diadelasemana{4}_Salida"
   IOField "Campo ES_23" at 479,311 size 86x32; FormatPattern 99999999999999999999
      ProcessValue <- "Planchadora1_Supervisores{2}_Diadelasemana{5}_Entrda"
   IOField "Campo ES_24" at 589,311 size 86x32; FormatPattern 99999999999999999999
      ProcessValue <- "Planchadora1_Supervisores{2}_Diadelasemana{5}_Salida"
   IOField "Campo ES_25" at 479,357 size 86x32; FormatPattern 99999999999999999999
      ProcessValue <- "Planchadora1_Supervisores{2}_Diadelasemana{6}_Entrda"
   IOField "Campo ES_26" at 589,357 size 86x32; FormatPattern 99999999999999999999
      ProcessValue <- "Planchadora1_Supervisores{2}_Diadelasemana{6}_Salida"
   IOField "Campo ES_27" at 479,403 size 86x32; FormatPattern 99999999999999999999
      ProcessValue <- "Planchadora1_Supervisores{2}_Diadelasemana{7}_Entrda"
   IOField "Campo ES_28" at 589,403 size 86x32; FormatPattern 99999999999999999999
      ProcessValue <- "Planchadora1_Supervisores{2}_Diadelasemana{7}_Salida"
   IOField "Campo ES_29" at 778,447 size 86x32; FormatPattern 99999999999999999999
      ProcessValue <- "Planchadora1_Supervisores{3}_Diadelasemana{1}_Entrda"
   IOField "Campo ES_30" at 885,447 size 86x32; FormatPattern 99999999999999999999
      ProcessValue <- "Planchadora1_Supervisores{3}_Diadelasemana{1}_Salida"
   IOField "Campo ES_31" at 778,173 size 86x32; FormatPattern 99999999999999999999
      ProcessValue <- "Planchadora1_Supervisores{3}_Diadelasemana{2}_Entrda"
   IOField "Campo ES_32" at 885,173 size 86x32; FormatPattern 99999999999999999999
      ProcessValue <- "Planchadora1_Supervisores{3}_Diadelasemana{2}_Salida"
   IOField "Campo ES_33" at 778,219 size 86x32; FormatPattern 99999999999999999999
      ProcessValue <- "Planchadora1_Supervisores{3}_Diadelasemana{3}_Entrda"
   IOField "Campo ES_34" at 885,219 size 86x32; FormatPattern 99999999999999999999
      ProcessValue <- "Planchadora1_Supervisores{3}_Diadelasemana{3}_Salida"
   IOField "Campo ES_35" at 778,265 size 86x32; FormatPattern 99999999999999999999
      ProcessValue <- "Planchadora1_Supervisores{3}_Diadelasemana{4}_Entrda"
   IOField "Campo ES_36" at 885,265 size 86x32; FormatPattern 99999999999999999999
      ProcessValue <- "Planchadora1_Supervisores{3}_Diadelasemana{4}_Salida"
   IOField "Campo ES_37" at 778,311 size 86x32; FormatPattern 99999999999999999999
      ProcessValue <- "Planchadora1_Supervisores{3}_Diadelasemana{5}_Entrda"
   IOField "Campo ES_38" at 885,311 size 86x32; FormatPattern 99999999999999999999
      ProcessValue <- "Planchadora1_Supervisores{3}_Diadelasemana{5}_Salida"
   IOField "Campo ES_39" at 778,357 size 86x32; FormatPattern 99999999999999999999
      ProcessValue <- "Planchadora1_Supervisores{3}_Diadelasemana{6}_Entrda"
   IOField "Campo ES_40" at 885,357 size 86x32; FormatPattern 99999999999999999999
      ProcessValue <- "Planchadora1_Supervisores{3}_Diadelasemana{6}_Salida"
   IOField "Campo ES_41" at 778,403 size 86x32; FormatPattern 99999999999999999999
      ProcessValue <- "Planchadora1_Supervisores{3}_Diadelasemana{7}_Entrda"
   IOField "Campo ES_42" at 885,403 size 86x32; FormatPattern 99999999999999999999
      ProcessValue <- "Planchadora1_Supervisores{3}_Diadelasemana{7}_Salida"
   TextField "Campo de texto_1" at 19,172 size 74x32; Text 'Lunes'
   TextField "Campo de texto_2" at 19,218 size 86x32; Text 'Martes'
   TextField "Campo de texto_3" at 19,264 size 116x32; Text 'Miercoles'
   TextField "Campo de texto_4" at 19,310 size 85x32; Text 'Jueves'
   TextField "Campo de texto_5" at 19,356 size 93x32; Text 'Viernes'
   TextField "Campo de texto_6" at 19,402 size 91x32; Text 'Sábado'
   TextField "Campo de texto_7" at 19,448 size 108x32; Text 'Domingo'
   TextField "Campo de texto_8" at 193,135 size 15x22; Text 'Text'
   TextField "Campo de texto_9" at 197,135 size 71x32; Text 'Inicio'
   TextField "Campo de texto_10" at 313,135 size 40x32; Text 'Fin'
   TextField "Campo de texto_11" at 486,135 size 15x22; Text 'Text'
   TextField "Campo de texto_12" at 490,135 size 71x32; Text 'Inicio'
   TextField "Campo de texto_13" at 606,135 size 40x32; Text 'Fin'
   TextField "Campo de texto_14" at 787,135 size 15x22; Text 'Text'
   TextField "Campo de texto_15" at 791,135 size 71x32; Text 'Inicio'
   TextField "Campo de texto_16" at 907,135 size 40x32; Text 'Fin'
   TextField "Campo de texto_18" at 182,50 size 200x32; Text 'Supervisor Nro 1'
   TextField "Campo de texto_19" at 474,49 size 200x32; Text 'Supervisor Nro 2'
   TextField "Campo de texto_20" at 775,48 size 200x32; Text 'Supervisor Nro 3'
   IOField "Campo ES_47" at 1066,447 size 86x32; FormatPattern 99999999999999999999
      ProcessValue <- "Planchadora1_Supervisores{4}_Diadelasemana{1}_Entrada"
   IOField "Campo ES_48" at 1171,447 size 86x32; FormatPattern 99999999999999999999
      ProcessValue <- "Planchadora1_Supervisores{4}_Diadelasemana{1}_Salida"
   IOField "Campo ES_49" at 1066,173 size 86x32; FormatPattern 99999999999999999999
      ProcessValue <- "Planchadora1_Supervisores{4}_Diadelasemana{2}_Entrada"
   IOField "Campo ES_50" at 1171,173 size 86x32; FormatPattern 99999999999999999999
      ProcessValue <- "Planchadora1_Supervisores{4}_Diadelasemana{2}_Salida"
   IOField "Campo ES_51" at 1066,219 size 86x32; FormatPattern 99999999999999999999
      ProcessValue <- "Planchadora1_Supervisores{4}_Diadelasemana{3}_Entrada"
   IOField "Campo ES_52" at 1171,219 size 86x32; FormatPattern 99999999999999999999
      ProcessValue <- "Planchadora1_Supervisores{4}_Diadelasemana{3}_Salida"
   IOField "Campo ES_53" at 1066,265 size 86x32; FormatPattern 99999999999999999999
      ProcessValue <- "Planchadora1_Supervisores{4}_Diadelasemana{4}_Entrada"
   IOField "Campo ES_54" at 1171,265 size 86x32; FormatPattern 99999999999999999999
      ProcessValue <- "Planchadora1_Supervisores{4}_Diadelasemana{4}_Salida"
   IOField "Campo ES_55" at 1066,311 size 86x32; FormatPattern 99999999999999999999
      ProcessValue <- "Planchadora1_Supervisores{4}_Diadelasemana{5}_Entrada"
   IOField "Campo ES_56" at 1171,311 size 86x32; FormatPattern 99999999999999999999
      ProcessValue <- "Planchadora1_Supervisores{4}_Diadelasemana{5}_Salida"
   IOField "Campo ES_57" at 1066,357 size 86x32; FormatPattern 99999999999999999999
      ProcessValue <- "Planchadora1_Supervisores{4}_Diadelasemana{6}_Entrada"
   IOField "Campo ES_58" at 1171,357 size 86x32; FormatPattern 99999999999999999999
      ProcessValue <- "Planchadora1_Supervisores{4}_Diadelasemana{6}_Salida"
   IOField "Campo ES_59" at 1066,403 size 86x32; FormatPattern 99999999999999999999
      ProcessValue <- "Planchadora1_Supervisores{4}_Diadelasemana{7}_Entrada"
   IOField "Campo ES_60" at 1171,403 size 86x32; FormatPattern 99999999999999999999
      ProcessValue <- "Planchadora1_Supervisores{4}_Diadelasemana{7}_Salida"
   TextField "Campo de texto_22" at 1075,135 size 71x32; Text 'Inicio'
   TextField "Campo de texto_23" at 1191,135 size 40x32; Text 'Fin'
   TextField "Campo de texto_24" at 1065,48 size 200x32; Text 'Supervisor Nro 4'
   Button "Botón_2968" at 1056,593 size 247x63; TextOff 'ESTADO DE CONTADORES'
      on Click: ActivateScreen("EstadoContadores", 0)
   IOField "Campo ES_46" at 188,93 size 188x32; FormatPattern ????????????????????????????????????????????????????????????????????????????????
      ProcessValue <- "Supervisor_Name_1"
   IOField "Campo ES_61" at 480,93 size 188x32; FormatPattern ????????????????????????????????????????????????????????????????????????????????
      ProcessValue <- "Supervisor_Name_2"
   IOField "Campo ES_87" at 781,93 size 188x32; FormatPattern ????????????????????????????????????????????????????????????????????????????????
      ProcessValue <- "Supervisor_Name_3"
   IOField "Campo ES_88" at 1071,93 size 188x32; FormatPattern ????????????????????????????????????????????????????????????????????????????????
      ProcessValue <- "Supervisor_Name_4"
   Button "Botón_357412" at 25,89 size 85x49; TextOff 'Actualizar Nombres'
      on Click: "S201_ActualizarSupervisor"()
   Button "Botón_8" at 1045,720 size 161x48; TextOff 'PRINCIPAL'
      on Click: ActivateScreen("Principal", 0)

screen "EstadoContadores" 1366x768, template "Pulsadores"
   IOField "Campo ES_1" at 160,100 size 100x30; FormatPattern 999999999999999
      ProcessValue <- "Planchadora1_Supervisores{1}_Tiempo"
   IOField "Campo ES_2" at 270,100 size 100x30; FormatPattern 999999999999999
      ProcessValue <- "Planchadora1_Supervisores{1}_Produccion"
   IOField "Campo ES_3" at 380,100 size 100x30; FormatPattern 999999999999999
      ProcessValue <- "Planchadora1_Supervisores{1}_Rendimiento"
   IOField "Campo ES_4" at 160,140 size 100x30; FormatPattern 999999999999999
      ProcessValue <- "Planchadora1_Supervisores{2}_Tiempo"
   IOField "Campo ES_5" at 270,140 size 100x30; FormatPattern 999999999999999
      ProcessValue <- "Planchadora1_Supervisores{2}_Produccion"
   IOField "Campo ES_6" at 380,140 size 100x30; FormatPattern 999999999999999
      ProcessValue <- "Planchadora1_Supervisores{2}_Rendimiento"
   IOField "Campo ES_7" at 600,140 size 60x30; FormatPattern 1
      ProcessValue <- "Planchadora1_Supervisores{2}_Estado"
   IOField "Campo ES_8" at 600,100 size 60x30; FormatPattern 1
      ProcessValue <- "Planchadora1_Supervisores{1}_Estado"
   IOField "Campo ES_9" at 160,180 size 100x30; FormatPattern 999999999999999
      ProcessValue <- "Planchadora1_Supervisores{3}_Tiempo"
   IOField "Campo ES_10" at 270,180 size 100x30; FormatPattern 999999999999999
      ProcessValue <- "Planchadora1_Supervisores{3}_Produccion"
   IOField "Campo ES_11" at 380,180 size 100x30; FormatPattern 999999999999999
      ProcessValue <- "Planchadora1_Supervisores{3}_Rendimiento"
   IOField "Campo ES_12" at 600,180 size 60x30; FormatPattern 1
      ProcessValue <- "Planchadora1_Supervisores{3}_Estado"
   IOField "Campo ES_13" at 160,50 size 100x30; FormatPattern 999999999999999
      ProcessValue <- "Planchadora1_TiempoTotal"
   IOField "Campo ES_14" at 270,50 size 100x30; FormatPattern 999999999999999
      ProcessValue <- "Planchadora1_ProductividadTotal"
   IOField "Campo ES_15" at 380,50 size 100x30; FormatPattern 999999999999999
      ProcessValue <- "Planchadora1_RendimientoTotal"
   IOField "Campo ES_16" at 160,270 size 100x30; FormatPattern 999999999999999
      ProcessValue <- "Planchadora1_Operadores{1}_Tiempo"
   IOField "Campo ES_17" at 270,270 size 100x30; FormatPattern 999999999999999
      ProcessValue <- "Planchadora1_Operadores{1}_Produccion"
   IOField "Campo ES_18" at 380,270 size 100x30; FormatPattern 999999999999999
      ProcessValue <- "Planchadora1_Operadores{1}_Rendimiento"
   IOField "Campo ES_19" at 600,270 size 60x30; FormatPattern 1
      ProcessValue <- "Planchadora1_Operadores{1}_Estado"
   IOField "Campo ES_20" at 160,310 size 100x30; FormatPattern 999999999999999
      ProcessValue <- "Planchadora1_Operadores{2}_Tiempo"
   IOField "Campo ES_21" at 270,310 size 100x30; FormatPattern 999999999999999
      ProcessValue <- "Planchadora1_Operadores{2}_Produccion"
   IOField "Campo ES_22" at 380,310 size 100x30; FormatPattern 999999999999999
      ProcessValue <- "Planchadora1_Operadores{2}_Rendimiento"
   IOField "Campo ES_23" at 600,310 size 60x30; FormatPattern 1
      ProcessValue <- "Planchadora1_Operadores{2}_Estado"
   IOField "Campo ES_24" at 160,350 size 100x30; FormatPattern 999999999999999
      ProcessValue <- "Planchadora1_Operadores{3}_Tiempo"
   IOField "Campo ES_25" at 270,350 size 100x30; FormatPattern 999999999999999
      ProcessValue <- "Planchadora1_Operadores{3}_Produccion"
   IOField "Campo ES_26" at 380,350 size 100x30; FormatPattern 999999999999999
      ProcessValue <- "Planchadora1_Operadores{3}_Rendimiento"
   IOField "Campo ES_27" at 600,350 size 60x30; FormatPattern 1
      ProcessValue <- "Planchadora1_Operadores{3}_Estado"
   IOField "Campo ES_28" at 160,390 size 100x30; FormatPattern 999999999999999
      ProcessValue <- "Planchadora1_Operadores{4}_Tiempo"
   IOField "Campo ES_29" at 270,390 size 100x30; FormatPattern 999999999999999
      ProcessValue <- "Planchadora1_Operadores{4}_Produccion"
   IOField "Campo ES_30" at 380,390 size 100x30; FormatPattern 999999999999999
      ProcessValue <- "Planchadora1_Operadores{4}_Rendimiento"
   IOField "Campo ES_31" at 600,390 size 60x30; FormatPattern 1
      ProcessValue <- "Planchadora1_Operadores{4}_Estado"
   IOField "Campo ES_32" at 160,430 size 100x30; FormatPattern 999999999999999
      ProcessValue <- "Planchadora1_Operadores{5}_Tiempo"
   IOField "Campo ES_33" at 270,430 size 100x30; FormatPattern 999999999999999
      ProcessValue <- "Planchadora1_Operadores{5}_Produccion"
   IOField "Campo ES_34" at 380,430 size 100x30; FormatPattern 999999999999999
      ProcessValue <- "Planchadora1_Operadores{5}_Rendimiento"
   IOField "Campo ES_35" at 600,430 size 60x30; FormatPattern 1
      ProcessValue <- "Planchadora1_Operadores{5}_Estado"
   IOField "Campo ES_36" at 160,470 size 100x30; FormatPattern 999999999999999
      ProcessValue <- "Planchadora1_Operadores{6}_Tiempo"
   IOField "Campo ES_37" at 270,470 size 100x30; FormatPattern 999999999999999
      ProcessValue <- "Planchadora1_Operadores{6}_Produccion"
   IOField "Campo ES_38" at 380,470 size 100x30; FormatPattern 999999999999999
      ProcessValue <- "Planchadora1_Operadores{6}_Rendimiento"
   IOField "Campo ES_39" at 600,470 size 60x30; FormatPattern 1
      ProcessValue <- "Planchadora1_Operadores{6}_Estado"
   IOField "Campo ES_40" at 160,510 size 100x30; FormatPattern 999999999999999
      ProcessValue <- "Planchadora1_Operadores{7}_Tiempo"
   IOField "Campo ES_41" at 270,510 size 100x30; FormatPattern 999999999999999
      ProcessValue <- "Planchadora1_Operadores{7}_Produccion"
   IOField "Campo ES_42" at 380,510 size 100x30; FormatPattern 999999999999999
      ProcessValue <- "Planchadora1_Operadores{7}_Rendimiento"
   IOField "Campo ES_43" at 600,510 size 60x30; FormatPattern 1
      ProcessValue <- "Planchadora1_Operadores{7}_Estado"
   IOField "Campo ES_44" at 160,550 size 100x30; FormatPattern 999999999999999
      ProcessValue <- "Planchadora1_Operadores{8}_Tiempo"
   IOField "Campo ES_45" at 270,550 size 100x30; FormatPattern 999999999999999
      ProcessValue <- "Planchadora1_Operadores{8}_Produccion"
   IOField "Campo ES_46" at 380,550 size 100x30; FormatPattern 999999999999999
      ProcessValue <- "Planchadora1_Operadores{8}_Rendimiento"
   IOField "Campo ES_47" at 600,550 size 60x30; FormatPattern 1
      ProcessValue <- "Planchadora1_Operadores{8}_Estado"
   IOField "Campo ES_48" at 160,590 size 100x30; FormatPattern 999999999999999
      ProcessValue <- "Planchadora1_Operadores{9}_Tiempo"
   IOField "Campo ES_49" at 270,590 size 100x30; FormatPattern 999999999999999
      ProcessValue <- "Planchadora1_Operadores{9}_Produccion"
   IOField "Campo ES_50" at 380,590 size 100x30; FormatPattern 999999999999999
      ProcessValue <- "Planchadora1_Operadores{9}_Rendimiento"
   IOField "Campo ES_51" at 600,590 size 60x30; FormatPattern 1
      ProcessValue <- "Planchadora1_Operadores{9}_Estado"
   IOField "Campo ES_52" at 160,630 size 100x30; FormatPattern 999999999999999
      ProcessValue <- "Planchadora1_Operadores{10}_Tiempo"
   IOField "Campo ES_53" at 270,630 size 100x30; FormatPattern 999999999999999
      ProcessValue <- "Planchadora1_Operadores{10}_Produccion"
   IOField "Campo ES_54" at 380,630 size 100x30; FormatPattern 999999999999999
      ProcessValue <- "Planchadora1_Operadores{10}_Rendimiento"
   IOField "Campo ES_55" at 600,630 size 60x30; FormatPattern 1
      ProcessValue <- "Planchadora1_Operadores{10}_Estado"
   IOField "Campo ES_56" at 160,220 size 100x30; FormatPattern 999999999999999
      ProcessValue <- "Planchadora1_Supervisores{4}_Tiempo"
   IOField "Campo ES_57" at 270,220 size 100x30; FormatPattern 999999999999999
      ProcessValue <- "Planchadora1_Supervisores{4}_Produccion"
   IOField "Campo ES_58" at 380,220 size 100x30; FormatPattern 999999999999999
      ProcessValue <- "Planchadora1_Supervisores{4}_Rendimiento"
   IOField "Campo ES_59" at 600,220 size 60x30; FormatPattern 1
      ProcessValue <- "Planchadora1_Supervisores{4}_Estado"
   Button "Botón_158654" at 1210,670 size 142x42; TextOff 'HORARIOS'
      on Click: ActivateScreen("Horario_Supervisor", 0)
   TextField "Campo de texto_1" at 181,22 size 59x22; Text 'Tiempo'
   TextField "Campo de texto_2" at 276,22 size 88x22; Text 'Produccion'
   TextField "Campo de texto_3" at 381,22 size 99x22; Text 'Rendimiento'
   TextField "Campo de texto_4" at 603,22 size 55x22; Text 'Estado'
   TextField "Campo de texto_6" at 38,274 size 76x22; Text 'Operador'
   IOField "Campo ES_60" at 790,270 size 100x30; FormatPattern 999999999999999
      ProcessValue <- "Planchadora2_Operadores{1}_Tiempo"
   IOField "Campo ES_61" at 900,270 size 100x30; FormatPattern 999999999999999
      ProcessValue <- "Planchadora2_Operadores{1}_Produccion"
   IOField "Campo ES_62" at 1010,270 size 100x30; FormatPattern 999999999999999
      ProcessValue <- "Planchadora2_Operadores{1}_Rendimiento"
   IOField "Campo ES_63" at 1230,270 size 60x30; FormatPattern 1
      ProcessValue <- "Planchadora2_Operadores{1}_Estado"
   IOField "Campo ES_64" at 790,310 size 100x30; FormatPattern 999999999999999
      ProcessValue <- "Planchadora2_Operadores{2}_Tiempo"
   IOField "Campo ES_65" at 900,310 size 100x30; FormatPattern 999999999999999
      ProcessValue <- "Planchadora2_Operadores{2}_Produccion"
   IOField "Campo ES_66" at 1010,310 size 100x30; FormatPattern 999999999999999
      ProcessValue <- "Planchadora2_Operadores{2}_Rendimiento"
   IOField "Campo ES_67" at 1230,310 size 60x30; FormatPattern 1
      ProcessValue <- "Planchadora2_Operadores{2}_Estado"
   IOField "Campo ES_68" at 790,350 size 100x30; FormatPattern 999999999999999
      ProcessValue <- "Planchadora2_Operadores{3}_Tiempo"
   IOField "Campo ES_69" at 900,350 size 100x30; FormatPattern 999999999999999
      ProcessValue <- "Planchadora2_Operadores{3}_Produccion"
   IOField "Campo ES_70" at 1010,350 size 100x30; FormatPattern 999999999999999
      ProcessValue <- "Planchadora2_Operadores{3}_Rendimiento"
   IOField "Campo ES_71" at 1230,350 size 60x30; FormatPattern 1
      ProcessValue <- "Planchadora2_Operadores{3}_Estado"
   IOField "Campo ES_72" at 790,390 size 100x30; FormatPattern 999999999999999
      ProcessValue <- "Planchadora2_Operadores{4}_Tiempo"
   IOField "Campo ES_73" at 900,390 size 100x30; FormatPattern 999999999999999
      ProcessValue <- "Planchadora2_Operadores{4}_Produccion"
   IOField "Campo ES_74" at 1010,390 size 100x30; FormatPattern 999999999999999
      ProcessValue <- "Planchadora2_Operadores{4}_Rendimiento"
   IOField "Campo ES_75" at 1230,390 size 60x30; FormatPattern 1
      ProcessValue <- "Planchadora2_Operadores{4}_Estado"
   IOField "Campo ES_76" at 790,430 size 100x30; FormatPattern 999999999999999
      ProcessValue <- "Planchadora2_Operadores{5}_Tiempo"
   IOField "Campo ES_77" at 900,430 size 100x30; FormatPattern 999999999999999
      ProcessValue <- "Planchadora2_Operadores{5}_Produccion"
   IOField "Campo ES_78" at 1010,430 size 100x30; FormatPattern 999999999999999
      ProcessValue <- "Planchadora2_Operadores{5}_Rendimiento"
   IOField "Campo ES_79" at 1230,430 size 60x30; FormatPattern 1
      ProcessValue <- "Planchadora2_Operadores{5}_Estado"
   IOField "Campo ES_80" at 790,470 size 100x30; FormatPattern 999999999999999
      ProcessValue <- "Planchadora2_Operadores{6}_Tiempo"
   IOField "Campo ES_81" at 900,470 size 100x30; FormatPattern 999999999999999
      ProcessValue <- "Planchadora2_Operadores{6}_Produccion"
   IOField "Campo ES_82" at 1010,470 size 100x30; FormatPattern 999999999999999
      ProcessValue <- "Planchadora2_Operadores{6}_Rendimiento"
   IOField "Campo ES_83" at 1230,470 size 60x30; FormatPattern 1
      ProcessValue <- "Planchadora2_Operadores{6}_Estado"
   IOField "Campo ES_84" at 790,510 size 100x30; FormatPattern 999999999999999
      ProcessValue <- "Planchadora2_Operadores{7}_Tiempo"
   IOField "Campo ES_85" at 900,510 size 100x30; FormatPattern 999999999999999
      ProcessValue <- "Planchadora2_Operadores{7}_Produccion"
   IOField "Campo ES_86" at 1010,510 size 100x30; FormatPattern 999999999999999
      ProcessValue <- "Planchadora2_Operadores{7}_Rendimiento"
   IOField "Campo ES_87" at 1230,510 size 60x30; FormatPattern 1
      ProcessValue <- "Planchadora2_Operadores{7}_Estado"
   IOField "Campo ES_88" at 790,550 size 100x30; FormatPattern 999999999999999
      ProcessValue <- "Planchadora2_Operadores{8}_Tiempo"
   IOField "Campo ES_89" at 900,550 size 100x30; FormatPattern 999999999999999
      ProcessValue <- "Planchadora2_Operadores{8}_Produccion"
   IOField "Campo ES_90" at 1010,550 size 100x30; FormatPattern 999999999999999
      ProcessValue <- "Planchadora2_Operadores{8}_Rendimiento"
   IOField "Campo ES_91" at 1230,550 size 60x30; FormatPattern 1
      ProcessValue <- "Planchadora2_Operadores{8}_Estado"
   IOField "Campo ES_92" at 790,590 size 100x30; FormatPattern 999999999999999
      ProcessValue <- "Planchadora2_Operadores{9}_Tiempo"
   IOField "Campo ES_93" at 900,590 size 100x30; FormatPattern 999999999999999
      ProcessValue <- "Planchadora2_Operadores{9}_Produccion"
   IOField "Campo ES_94" at 1010,590 size 100x30; FormatPattern 999999999999999
      ProcessValue <- "Planchadora2_Operadores{9}_Rendimiento"
   IOField "Campo ES_95" at 1230,590 size 60x30; FormatPattern 1
      ProcessValue <- "Planchadora2_Operadores{9}_Estado"
   IOField "Campo ES_96" at 790,630 size 100x30; FormatPattern 999999999999999
      ProcessValue <- "Planchadora2_Operadores{10}_Tiempo"
   IOField "Campo ES_97" at 900,630 size 100x30; FormatPattern 999999999999999
      ProcessValue <- "Planchadora2_Operadores{10}_Produccion"
   IOField "Campo ES_98" at 1010,630 size 100x30; FormatPattern 999999999999999
      ProcessValue <- "Planchadora2_Operadores{10}_Rendimiento"
   IOField "Campo ES_99" at 1230,630 size 60x30; FormatPattern 1
      ProcessValue <- "Planchadora2_Operadores{10}_Estado"
   IOField "Campo ES_100" at 790,100 size 100x30; FormatPattern 999999999999999
      ProcessValue <- "Planchadora2_Supervisores{1}_Tiempo"
   IOField "Campo ES_101" at 900,100 size 100x30; FormatPattern 999999999999999
      ProcessValue <- "Planchadora2_Supervisores{1}_Produccion"
   IOField "Campo ES_102" at 1010,100 size 100x30; FormatPattern 999999999999999
      ProcessValue <- "Planchadora2_Supervisores{1}_Rendimiento"
   IOField "Campo ES_103" at 1230,100 size 60x30; FormatPattern 1
      ProcessValue <- "Planchadora2_Supervisores{1}_Estado"
   IOField "Campo ES_104" at 790,140 size 100x30; FormatPattern 999999999999999
      ProcessValue <- "Planchadora2_Supervisores{2}_Tiempo"
   IOField "Campo ES_105" at 900,140 size 100x30; FormatPattern 999999999999999
      ProcessValue <- "Planchadora2_Supervisores{2}_Produccion"
   IOField "Campo ES_106" at 1010,140 size 100x30; FormatPattern 999999999999999
      ProcessValue <- "Planchadora2_Supervisores{2}_Rendimiento"
   IOField "Campo ES_107" at 1230,140 size 60x30; FormatPattern 1
      ProcessValue <- "Planchadora2_Supervisores{2}_Estado"
   IOField "Campo ES_108" at 790,180 size 100x30; FormatPattern 999999999999999
      ProcessValue <- "Planchadora2_Supervisores{3}_Tiempo"
   IOField "Campo ES_109" at 900,180 size 100x30; FormatPattern 999999999999999
      ProcessValue <- "Planchadora2_Supervisores{3}_Produccion"
   IOField "Campo ES_110" at 1010,180 size 100x30; FormatPattern 999999999999999
      ProcessValue <- "Planchadora2_Supervisores{3}_Rendimiento"
   IOField "Campo ES_111" at 1230,180 size 60x30; FormatPattern 1
      ProcessValue <- "Planchadora2_Supervisores{3}_Estado"
   IOField "Campo ES_112" at 790,220 size 100x30; FormatPattern 999999999999999
      ProcessValue <- "Planchadora2_Supervisores{4}_Tiempo"
   IOField "Campo ES_113" at 900,220 size 100x30; FormatPattern 999999999999999
      ProcessValue <- "Planchadora2_Supervisores{4}_Produccion"
   IOField "Campo ES_114" at 1010,220 size 100x30; FormatPattern 999999999999999
      ProcessValue <- "Planchadora2_Supervisores{4}_Rendimiento"
   IOField "Campo ES_115" at 1230,220 size 60x30; FormatPattern 1
      ProcessValue <- "Planchadora2_Supervisores{4}_Estado"
   IOField "Campo ES_116" at 790,50 size 100x30; FormatPattern 999999999999999
      ProcessValue <- "Planchadora2_TiempoTotal"
   IOField "Campo ES_117" at 900,50 size 100x30; FormatPattern 999999999999999
      ProcessValue <- "Planchadora2_ProductividadTotal"
   IOField "Campo ES_118" at 1010,50 size 100x30; FormatPattern 999999999999999
      ProcessValue <- "Planchadora2_RendimientoTotal"
   TextField "Campo de texto_5" at 33,104 size 87x22; Text 'Supervisor'
   TextField "Campo de texto_16" at 27,54 size 98x22; Text 'Planchadora'
   TextField "Campo de texto_17" at 131,104 size 15x22; Text '1'
   TextField "Campo de texto_18" at 131,144 size 15x22; Text '2'
   TextField "Campo de texto_19" at 131,184 size 15x22; Text '3'
   TextField "Campo de texto_20" at 131,224 size 15x22; Text '4'
   TextField "Campo de texto_7" at 131,274 size 15x22; Text '1'
   TextField "Campo de texto_8" at 131,314 size 15x22; Text '2'
   TextField "Campo de texto_9" at 131,354 size 15x22; Text '3'
   TextField "Campo de texto_10" at 131,394 size 15x22; Text '4'
   TextField "Campo de texto_11" at 131,434 size 15x22; Text '5'
   TextField "Campo de texto_12" at 131,474 size 15x22; Text '6'
   TextField "Campo de texto_13" at 131,514 size 15x22; Text '7'
   TextField "Campo de texto_14" at 131,554 size 15x22; Text '8'
   TextField "Campo de texto_15" at 131,594 size 15x22; Text '9'
   TextField "Campo de texto_21" at 131,634 size 25x22; Text '10'
   TextField "Campo de texto_22" at 755,274 size 15x22; Text '1'
   TextField "Campo de texto_23" at 755,314 size 15x22; Text '2'
   TextField "Campo de texto_24" at 755,354 size 15x22; Text '3'
   TextField "Campo de texto_25" at 755,394 size 15x22; Text '4'
   TextField "Campo de texto_26" at 755,434 size 15x22; Text '5'
   TextField "Campo de texto_27" at 755,474 size 15x22; Text '6'
   TextField "Campo de texto_28" at 755,514 size 15x22; Text '7'
   TextField "Campo de texto_29" at 755,554 size 15x22; Text '8'
   TextField "Campo de texto_30" at 755,594 size 15x22; Text '9'
   TextField "Campo de texto_31" at 755,634 size 25x22; Text '10'
   TextField "Campo de texto_32" at 131,56 size 15x22; Text '1'
   TextField "Campo de texto_33" at 755,104 size 15x22; Text '1'
   TextField "Campo de texto_34" at 755,144 size 15x22; Text '2'
   TextField "Campo de texto_35" at 755,184 size 15x22; Text '3'
   TextField "Campo de texto_36" at 755,224 size 15x22; Text '4'
   TextField "Campo de texto_37" at 755,56 size 15x22; Text '2'
   TextField "Campo de texto_38" at 811,22 size 59x22; Text 'Tiempo'
   TextField "Campo de texto_39" at 906,22 size 88x22; Text 'Produccion'
   TextField "Campo de texto_40" at 1011,22 size 99x22; Text 'Rendimiento'
   TextField "Campo de texto_41" at 1233,22 size 55x22; Text 'Estado'
   IOField "Campo ES_119" at 490,100 size 100x30; FormatPattern 999999999999999
      ProcessValue <- "Planchadora1_Supervisores{1}_RendPesado"
   IOField "Campo ES_120" at 490,140 size 100x30; FormatPattern 999999999999999
      ProcessValue <- "Planchadora1_Supervisores{2}_RendPesado"
   IOField "Campo ES_121" at 490,180 size 100x30; FormatPattern 999999999999999
      ProcessValue <- "Planchadora1_Supervisores{3}_RendPesado"
   IOField "Campo ES_122" at 490,50 size 100x30; FormatPattern 999999999999999
      ProcessValue <- "Planchadora1_RendPesado"
   IOField "Campo ES_123" at 490,270 size 100x30; FormatPattern 999999999999999
      ProcessValue <- "Planchadora1_Operadores{1}_RendPesado"
   IOField "Campo ES_124" at 490,310 size 100x30; FormatPattern 999999999999999
      ProcessValue <- "Planchadora1_Operadores{2}_RendPesado"
   IOField "Campo ES_125" at 490,350 size 100x30; FormatPattern 999999999999999
      ProcessValue <- "Planchadora1_Operadores{3}_RendPesado"
   IOField "Campo ES_126" at 490,390 size 100x30; FormatPattern 999999999999999
      ProcessValue <- "Planchadora1_Operadores{4}_RendPesado"
   IOField "Campo ES_127" at 490,430 size 100x30; FormatPattern 999999999999999
      ProcessValue <- "Planchadora1_Operadores{5}_RendPesado"
   IOField "Campo ES_128" at 490,470 size 100x30; FormatPattern 999999999999999
      ProcessValue <- "Planchadora1_Operadores{6}_RendPesado"
   IOField "Campo ES_129" at 490,510 size 100x30; FormatPattern 999999999999999
      ProcessValue <- "Planchadora1_Operadores{7}_RendPesado"
   IOField "Campo ES_130" at 490,550 size 100x30; FormatPattern 999999999999999
      ProcessValue <- "Planchadora1_Operadores{8}_RendPesado"
   IOField "Campo ES_131" at 490,590 size 100x30; FormatPattern 999999999999999
      ProcessValue <- "Planchadora1_Operadores{9}_RendPesado"
   IOField "Campo ES_132" at 490,630 size 100x30; FormatPattern 999999999999999
      ProcessValue <- "Planchadora1_Operadores{10}_RendPesado"
   IOField "Campo ES_133" at 490,220 size 100x30; FormatPattern 999999999999999
      ProcessValue <- "Planchadora1_Supervisores{4}_RendPesado"
   TextField "Campo de texto_42" at 491,22 size 99x22; Text 'Rendimiento'
   IOField "Campo ES_134" at 1120,100 size 100x30; FormatPattern 999999999999999
      ProcessValue <- "Planchadora2_Supervisores{1}_RendPesado"
   IOField "Campo ES_135" at 1120,140 size 100x30; FormatPattern 999999999999999
      ProcessValue <- "Planchadora2_Supervisores{2}_RendPesado"
   IOField "Campo ES_136" at 1120,180 size 100x30; FormatPattern 999999999999999
      ProcessValue <- "Planchadora2_Supervisores{3}_RendPesado"
   IOField "Campo ES_137" at 1120,50 size 100x30; FormatPattern 999999999999999
      ProcessValue <- "Planchadora2_RendPesado"
   IOField "Campo ES_138" at 1120,270 size 100x30; FormatPattern 999999999999999
      ProcessValue <- "Planchadora2_Operadores{1}_RendPesado"
   IOField "Campo ES_139" at 1120,310 size 100x30; FormatPattern 999999999999999
      ProcessValue <- "Planchadora2_Operadores{2}_RendPesado"
   IOField "Campo ES_140" at 1120,350 size 100x30; FormatPattern 999999999999999
      ProcessValue <- "Planchadora2_Operadores{3}_RendPesado"
   IOField "Campo ES_141" at 1120,390 size 100x30; FormatPattern 999999999999999
      ProcessValue <- "Planchadora2_Operadores{4}_RendPesado"
   IOField "Campo ES_142" at 1120,430 size 100x30; FormatPattern 999999999999999
      ProcessValue <- "Planchadora2_Operadores{5}_RendPesado"
   IOField "Campo ES_143" at 1120,470 size 100x30; FormatPattern 999999999999999
      ProcessValue <- "Planchadora2_Operadores{6}_RendPesado"
   IOField "Campo ES_144" at 1120,510 size 100x30; FormatPattern 999999999999999
      ProcessValue <- "Planchadora2_Operadores{7}_RendPesado"
   IOField "Campo ES_145" at 1120,550 size 100x30; FormatPattern 999999999999999
      ProcessValue <- "Planchadora2_Operadores{8}_RendPesado"
   IOField "Campo ES_146" at 1120,590 size 100x30; FormatPattern 999999999999999
      ProcessValue <- "Planchadora2_Operadores{9}_RendPesado"
   IOField "Campo ES_147" at 1120,630 size 100x30; FormatPattern 999999999999999
      ProcessValue <- "Planchadora2_Operadores{10}_RendPesado"
   IOField "Campo ES_148" at 1120,220 size 100x30; FormatPattern 999999999999999
      ProcessValue <- "Planchadora2_Supervisores{4}_RendPesado"
   TextField "Campo de texto_43" at 1121,22 size 99x22; Text 'Rendimiento'
   Button "Botón_8" at 1045,720 size 161x48; TextOff 'PRINCIPAL'
      on Click: ActivateScreen("Principal", 0)

screen "Tendencias" 1366x768, template "Pulsadores"
   TextField "Campo de texto_2" at 281,6 size 751x47; Text 'OBJETIVO Y RENDIMIENTO ACUMULADO'
   Button "Botón_8" at 1045,720 size 161x48; TextOff 'PRINCIPAL'
      on Click: ActivateScreen("Principal", 0)
   TrendView "Visor de curvas_1" at 20,54 size 1322x641
   Button "Botón_26" at 725,720 size 161x48; TextOff 'Tendencias PL1'
      on Click: ActivateScreen("Tendencias", 0)
   Button "Botón_27" at 885,720 size 161x48; TextOff 'Tendencias PL2'
      on Click: ActivateScreen("TendenciasPL2", 0)

screen "TendenciasPL2" 1366x768, template "Pulsadores"
   TrendView "Visor de curvas_1" at 6,30 size 1338x318
   TrendView "Visor de curvas_2" at 6,394 size 1338x318
   TextField "Campo de texto_1" at 341,360 size 668x31; Text 'PRODUCTIVIDAD Y RENDIMIENTO CADA 15Min PLANCHA 2'
   TextField "Campo de texto_2" at 269,0 size 813x31; Text 'PRODUCTIVIDAD Y RENDIMIENTO ACUMULADO POR TURNO PLANCHA 2'
   Button "Botón_8" at 1045,720 size 161x48; TextOff 'PRINCIPAL'
      on Click: ActivateScreen("Principal", 0)

screen "Alarmas" 1366x768, template "Pulsadores"
   AlarmView "Visor de avisos_1" at 11,46 size 1340x310
   AlarmView "Visor de avisos_2" at 11,419 size 1340x274
   TextField "Campo de texto_3" at 537,8 size 232x35; Text 'Alarmas Actuales'
   TextField "Campo de texto_1" at 515,376 size 276x35; Text 'Historico de Alarmas'
   Button "Botón_250" at 1045,720 size 161x48; TextOff 'PRINCIPAL'
      on Click: ActivateScreen("Principal", 0)

screen "RegyClientes" 1366x768, template "Pulsadores"
   IOField "Campo ES_46" at 1034,6 size 249x37; FormatPattern 9999999999999999999999999999999999999999
      ProcessValue <- "Planchadora1_FechaHoraPLC"
   Button "Botón_5423" at 756,90 size 88x32; TextOff 'Crear'
      on Click: "S101_EscribirCliente"()
   IOField "Campo ES_2" at 506,90 size 236x32; FormatPattern ????????????????????????????????????????????????????????????????????????????????
      ProcessValue <- "Name_Nuevo"
   IOField "Campo ES_3" at 442,90 size 60x32; FormatPattern 99
      ProcessValue <- "ID_Nuevo"
   TextField "Campo de texto_1" at 445,62 size 122x22; Text 'Agregar Cliente'
   Button "Botón_1578" at 756,162 size 88x32; TextOff 'Actualizar'
      on Click: "S102_CambiarCliente"()
   IOField "Campo ES_1" at 506,162 size 236x32; FormatPattern ????????????????????????????????????????????????????????????????????????????????
      ProcessValue <- "Name_Cambiar"
   IOField "Campo ES_4" at 442,162 size 60x32; FormatPattern 99
      ProcessValue <- "ID_Cambiar"
   TextField "Campo de texto_2" at 445,134 size 133x22; Text 'Modificar Cliente'
   IOField "Campo ES_5" at 98,59 size 252x32; FormatPattern ??????????????????????????????????????????????????????????????????????????????????????????????????????????????????????????????????????????????????????????????????????????????????????????????????????????????????????????????????????????????????????????????
      ProcessValue <- "Name_1"
   IOField "Campo ES_6" at 34,59 size 60x32; FormatPattern 99
      ProcessValue <- "ID_1"
   IOField "Campo ES_7" at 98,91 size 252x32; FormatPattern ??????????????????????????????????????????????????????????????????????????????????????????????????????????????????????????????????????????????????????????????????????????????????????????????????????????????????????????????????????????????????????????????
      ProcessValue <- "Name_2"
   IOField "Campo ES_8" at 34,91 size 60x32; FormatPattern 99
      ProcessValue <- "ID_2"
   IOField "Campo ES_9" at 98,123 size 252x32; FormatPattern ??????????????????????????????????????????????????????????????????????????????????????????????????????????????????????????????????????????????????????????????????????????????????????????????????????????????????????????????????????????????????????????????
      ProcessValue <- "Name_3"
   IOField "Campo ES_10" at 34,123 size 60x32; FormatPattern 99
      ProcessValue <- "ID_3"
   IOField "Campo ES_11" at 98,155 size 252x32; FormatPattern ????????????????????????????????????????????????????????????????????????????????
      ProcessValue <- "Name_4"
   IOField "Campo ES_12" at 34,155 size 60x32; FormatPattern 99
      ProcessValue <- "ID_4"
   IOField "Campo ES_13" at 98,187 size 252x32; FormatPattern ????????????????????????????????????????????????????????????????????????????????
      ProcessValue <- "Name_5"
   IOField "Campo ES_14" at 34,187 size 60x32; FormatPattern 99
      ProcessValue <- "ID_5"
   Button "Botón_4" at 300,22 size 96x32; TextOff 'Actualizar'
      on Click: SetTag("ID_1", 1); "S103_ActualizarLista"()
   Button "Botón_7" at 1100,259 size 96x32; TextOff 'Actualizar'
      on Click: "S200_CambSupervisor"()
   IOField "Campo ES_25" at 1166,221 size 188x32; FormatPattern ????????????????????????????????????????????????????????????????????????????????
      ProcessValue <- "Supervisor_Camb"
   IOField "Campo ES_26" at 1100,221 size 60x32; FormatPattern 9
      ProcessValue <- "Supervisor_ID_Camb"
   TextField "Campo de texto_3" at 1101,196 size 123x22; Text 'Modificar Turno'
   IOField "Campo ES_27" at 899,230 size 188x32; FormatPattern ????????????????????????????????????????????????????????????????????????????????
      ProcessValue <- "Supervisor_Name_1"
   IOField "Campo ES_29" at 899,262 size 188x32; FormatPattern ????????????????????????????????????????????????????????????????????????????????
      ProcessValue <- "Supervisor_Name_2"
   IOField "Campo ES_31" at 899,294 size 188x32; FormatPattern ????????????????????????????????????????????????????????????????????????????????
      ProcessValue <- "Supervisor_Name_3"
   IOField "Campo ES_33" at 899,326 size 188x32; FormatPattern ????????????????????????????????????????????????????????????????????????????????
      ProcessValue <- "Supervisor_Name_4"
   TextField "Campo de texto_4" at 73,22 size 116x31; Text 'CLIENTES'
   TextField "Campo de texto_5" at 890,193 size 81x31; Text 'Turnos'
   TextField "Campo de texto_6" at 871,233 size 16x26; Text '1'
   TextField "Campo de texto_7" at 871,265 size 16x26; Text '2'
   TextField "Campo de texto_8" at 871,297 size 16x26; Text '3'
   TextField "Campo de texto_9" at 871,329 size 16x26; Text '4'
   IOField "Campo ES_15" at 506,330 size 236x32; FormatPattern ????????????????????????????????????????????????????????????????????????????????
      ProcessValue <- "Name_OP_Nuevo"
   IOField "Campo ES_16" at 442,330 size 60x32; FormatPattern 99
      ProcessValue <- "ID_OP_Nuevo"
   TextField "Campo de texto_10" at 445,302 size 140x22; Text 'Agregar Operador'
   IOField "Campo ES_17" at 506,402 size 236x32; FormatPattern ????????????????????????????????????????????????????????????????????????????????
      ProcessValue <- "Name_OP_Cambiar"
   IOField "Campo ES_18" at 442,402 size 60x32; FormatPattern 99
      ProcessValue <- "ID_OP_Cambiar"
   TextField "Campo de texto_11" at 445,374 size 151x22; Text 'Modificar Operador'
   IOField "Campo ES_19" at 98,299 size 252x32; FormatPattern ??????????????????????????????????????????????????????????????????????????????????????????????????????????????????????????????????????????????????????????????????????????????????????????????????????????????????????????????????????????????????????????????
      ProcessValue <- "Name_OP_1"
   IOField "Campo ES_20" at 34,299 size 60x32; FormatPattern 99
      ProcessValue <- "ID_OP_1"
   IOField "Campo ES_21" at 98,331 size 252x32; FormatPattern ??????????????????????????????????????????????????????????????????????????????????????????????????????????????????????????????????????????????????????????????????????????????????????????????????????????????????????????????????????????????????????????????
      ProcessValue <- "Name_OP_2"
   IOField "Campo ES_22" at 34,331 size 60x32; FormatPattern 99
      ProcessValue <- "ID_OP_2"
   IOField "Campo ES_23" at 98,363 size 252x32; FormatPattern ??????????????????????????????????????????????????????????????????????????????????????????????????????????????????????????????????????????????????????????????????????????????????????????????????????????????????????????????????????????????????????????????
      ProcessValue <- "Name_OP_3"
   IOField "Campo ES_24" at 34,363 size 60x32; FormatPattern 99
      ProcessValue <- "ID_OP_3"
   IOField "Campo ES_28" at 98,395 size 252x32; FormatPattern ????????????????????????????????????????????????????????????????????????????????
      ProcessValue <- "Name_OP_4"
   IOField "Campo ES_30" at 34,395 size 60x32; FormatPattern 99
      ProcessValue <- "ID_OP_4"
   IOField "Campo ES_32" at 98,427 size 252x32; FormatPattern ????????????????????????????????????????????????????????????????????????????????
      ProcessValue <- "Name_OP_5"
   IOField "Campo ES_34" at 34,427 size 60x32; FormatPattern 99
      ProcessValue <- "ID_OP_5"
   Button "Botón_10" at 300,262 size 96x32; TextOff 'Actualizar'
      on Click: SetTag("ID_OP_1", 1); "S303_ActualizarListaOp"()
   TextField "Campo de texto_12" at 73,262 size 159x31; Text 'OPERADORES'
   Button "Botón_11" at 756,330 size 88x32; TextOff 'Crear'
      on Click: "S301_EscribirOperador"()
   Button "Botón_12" at 756,402 size 88x32; TextOff 'Actualizar'
      on Click: "S302_CambiarOperador"()
   Button "Botón_13" at 363,181 size 39x38; TextOff 'Text'
      on Click: function_dd21b452("ID_1", 1); "S103_ActualizarLista"()
   Button "Botón_14" at 363,59 size 39x38; TextOff 'Text'
      on Click: function_b9b71300("ID_1", 1); "S103_ActualizarLista"()
   Button "Botón_2" at 363,421 size 39x38; TextOff 'Text'
      on Click: function_dd21b452("ID_OP_1", 1); "S303_ActualizarListaOp"()
   Button "Botón_3" at 363,299 size 39x38; TextOff 'Text'
      on Click: function_b9b71300("ID_OP_1", 1); "S303_ActualizarListaOp"()
   Button "Botón_8" at 1045,720 size 161x48; TextOff 'PRINCIPAL'
      on Click: ActivateScreen("Principal", 0)
   Button "Botón_6" at 410,561 size 96x32; TextOff 'Crear'
      on Click: "I101_EscribirIndice"()
   IOField "Campo ES_35" at 320,561 size 76x32; FormatPattern 9999
      ProcessValue <- "Idx_Name_Nuevo"
   IOField "Campo ES_36" at 256,561 size 60x32; FormatPattern 99
      ProcessValue <- "Idx_ID_Nuevo"
   TextField "Campo de texto_13" at 259,537 size 138x22; Text 'AGREGAR INDICE'
   Button "Botón_9" at 410,633 size 96x32; TextOff 'Actualizar'
      on Click: "I102_CambiarIndice"()
   IOField "Campo ES_37" at 320,633 size 76x32; FormatPattern 9999
      ProcessValue <- "Idx_Name_Cambiar"
   IOField "Campo ES_38" at 256,633 size 60x32; FormatPattern 99
      ProcessValue <- "Idx_ID_Cambiar"
   TextField "Campo de texto_14" at 259,609 size 155x22; Text 'MODIFICAR INDICE'
   IOField "Campo ES_39" at 104,530 size 76x32; FormatPattern 9999
      ProcessValue <- "Idx_Name_1"
   IOField "Campo ES_40" at 40,530 size 60x32; FormatPattern 99
      ProcessValue <- "Idx_ID_1"
   IOField "Campo ES_41" at 104,562 size 76x32; FormatPattern 9999
      ProcessValue <- "Idx_Name_2"
   IOField "Campo ES_42" at 40,562 size 60x32; FormatPattern 99
      ProcessValue <- "Idx_ID_2"
   IOField "Campo ES_43" at 104,594 size 76x32; FormatPattern 9999
      ProcessValue <- "Idx_Name_3"
   IOField "Campo ES_44" at 40,594 size 60x32; FormatPattern 99
      ProcessValue <- "Idx_ID_3"
   IOField "Campo ES_45" at 104,626 size 76x32; FormatPattern 9999
      ProcessValue <- "Idx_Name_4"
   IOField "Campo ES_47" at 40,626 size 60x32; FormatPattern 99
      ProcessValue <- "Idx_ID_4"
   IOField "Campo ES_48" at 104,658 size 76x32; FormatPattern 9999
      ProcessValue <- "Idx_Name_5"
   IOField "Campo ES_49" at 40,658 size 60x32; FormatPattern 99
      ProcessValue <- "Idx_ID_5"
   Button "Botón_15" at 42,493 size 96x32; TextOff 'Actualizar'
      on Click: SetTag("Idx_ID_1", 1); "I103_ActualizarIndice"()
   TextField "Campo de texto_15" at 159,493 size 230x31; Text 'INDICES PLANCHAS'
   Button "Botón_16" at 185,652 size 39x38; TextOff 'Text'
      on Click: function_dd21b452("Idx_ID_1", 1); "I103_ActualizarIndice"()
   Button "Botón_17" at 185,530 size 39x38; TextOff 'Text'
      on Click: function_b9b71300("Idx_ID_1", 1); "I103_ActualizarIndice"()
   Button "Botón_18" at 1100,304 size 254x63; TextOff 'HORARIOS'
      on Press: ActivateScreen("Horario_Supervisor", 0)

screen "Configuracion" 1366x768, template "Pulsadores"
   Button "Botón_3" at 1046,326 size 96x63; TextOff 'Generar Informe Diario'
      on Click: "S07_InformeDiario_Planchas"(N)
   Button "Botón_4" at 996,425 size 170x42; TextOff 'Cerrar SCADA'
      on Click: StopRuntime(0)
   IOField "Campo ES_87" at 243,293 size 75x31; FormatPattern 99.999
      ProcessValue <- "Planchadora1_FactorCorrRend"
   TextField "Campo de texto_30" at 97,289 size 138x40; Text 'Factor Correccion Rendimiento'
   TextField "Campo de texto_31" at 41,298 size 34x22; Text 'PL1'
   IOField "Campo ES_46" at 134,201 size 185x31; FormatPattern 9999999999999999999999999999999999999999
      ProcessValue <- "Planchadora1_FechaHoraPLC"
   DateTimeField "Campo de fecha y hora_1" at 134,232 size 185x31
   TextField "Campo de texto_25" at 28,206 size 82x22; Text 'Fecha PLC'
   TextField "Campo de texto_26" at 33,237 size 73x22; Text 'Fecha PC'
   SymbolicIOField "Campo ES simbólico_1" at 336,201 size 136x31; TextOn '1'; TextOff '0'; TextList "Lista de textos_1"
      ProcessValue <- "Planchadora1_WeekDay"
   Button "Botón_5" at 494,201 size 96x63; TextOff 'Grabar Actuales Planchadora'
      on Click: "S03_Write_data_record_into_a_table"()
   TextField "Campo de texto_1" at 925,325 size 106x22; Text 'Planchadoras'
   AlarmView "Visor de avisos_1" at 2,15 size 1363x158
   IOField "Campo ES_7" at 243,341 size 75x31; FormatPattern 99.999
      ProcessValue <- "Planchadora2_FactorCorrRend"
   TextField "Campo de texto_3" at 97,337 size 138x40; Text 'Factor Correccion Rendimiento'
   TextField "Campo de texto_4" at 41,346 size 34x22; Text 'PL2'
   Button "Botón_11" at 387,288 size 277x42; TextOff 'LAVs 1 a 3'
      on Click: ActivateScreen("VariablesLavs", 0)
   Button "Botón_8" at 387,347 size 277x42; TextOff 'LAV 4'
      on Click: ActivateScreen("VariablesLavs_1", 0)
   Button "Botón_13" at 1024,248 size 169x47; TextOff 'Prog LAV 1'
      on Click: ActivateScreen("Prog_Lav1_0", 0)
   Button "Botón_2" at 1045,720 size 161x48; TextOff 'PRINCIPAL'
      on Click: ActivateScreen("Principal", 0)
   Button "Botón_1" at 430,450 size 96x32; TextOff 'Mensual'
      on Click: "S404_ActMes"(); "S500_InformePeriodico"(1, "Inf_Ano", "Inf_Mes")

